METHOD Reset_Done : BOOL
VAR
	sTemp1 : T_MaxString;
END_VAR
IF sData = '' THEN
	Reset_Done := FALSE;
ELSE
	sTemp1 := sData;
	IF FC_Check_SOH(sTemp1) AND FC_Check_ACK(sTemp1) AND FC_Check_EOT(sTemp1) AND FC_Check_R(sTemp1) THEN
		Reset_Done := TRUE;
	ELSE
		Reset_Done := FALSE;
	END_IF
END_IF
END_METHOD

METHOD Start : BOOL
// Description : Ask for the status of the machine
VAR_INPUT
END_VAR
VAR
	sTemp1 : STRING;
	sTemp2 : STRING;
END_VAR
sData := '';
sTemp1 := 'S';
sTemp2 := CONCAT(SOH, sTemp1);
sCmd := CONCAT(sTemp2, EOT);
THIS^.Send(sCmd);
END_METHOD

METHOD Start_Done : BOOL
VAR
	sTemp1 : T_MaxString;
END_VAR
IF sData = '' THEN
	Start_Done := FALSE;
ELSE
	sTemp1 := sData;
	IF FC_Check_SOH(sTemp1) AND FC_Check_ACK(sTemp1) AND FC_Check_EOT(sTemp1) AND FC_Check_S(sTemp1) THEN
		Start_Done := TRUE;
	ELSE
		Start_Done := FALSE;
	END_IF
END_IF
END_METHOD

END_FUNCTION_BLOCK

// ---- FBs/Ethernet/FB_EthDevice.TcPOU
FUNCTION_BLOCK FB_EthDevice
VAR_INPUT
	bEnable		: BOOL 			:= FALSE;				(* TRUE => enable client data exchange, FALSE => disable *)
	sSrvNetID	: T_AmsNetID	:= '';					(* TwinCAT TCP/IP server network address *)
	sRemoteHost	: T_IPv4Addr 	:= '127.0.0.1';			(* Server network address *)
	nRemotePort	: UDINT 		:= 200;					(* Server port number *)
	bLogEnable	: BOOL 			:= FALSE;				(* TRUE => Enable log message output, FALSE => Disable *)
	sLogPrefix	: STRING 		:= 'CLIENT::';			(* Log message description string (allows the identification of log message source) *)
END_VAR
VAR_OUTPUT
	sData						: T_MaxString;			(* Output received Data *)
	bConnected					: BOOL := FALSE;		(* TCP/IP connection state *)	
END_VAR
VAR
	fbConnection				: FB_ClientConnection;	(* Client connection/data exchange control function block *)
	fbTx 						: FB_FrameFifo;			(* Tx fifo *)
	fbRx 						: FB_FrameFifo;			(* Rx fifo *)
	
	sLogMessage					: T_MaxString;
	sTemData					: T_MaxString;			(* Output received Data *)
END_VAR

IF bConnected := fbConnection.bConnected THEN
	A_Receive();
END_IF

A_Call();

IF NOT fbConnection.RxBusy THEN
	sData := sTemData;
END_IF

ACTION A_Call:
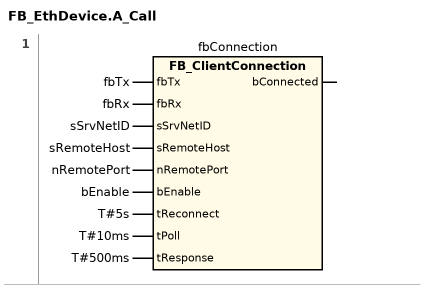
// NETWORK 1
fbConnection(
    fbTx := fbTx,
    fbRx := fbRx,
    sSrvNetID := sSrvNetID,
    sRemoteHost := sRemoteHost,
    nRemotePort := nRemotePort,
    bEnable := bEnable,
    tReconnect := T#5s,
    tPoll := T#10ms,
    tResponse := T#500ms); // FB_ClientConnection
END_ACTION

ACTION A_Receive:
	(*--------------------- Get received message strings --------------------------------*)
	REPEAT
		fbRx.RemoveHead( );(* Fetch string from rx fifo *)
		IF fbRx.bOk THEN(* Success *)
	
		(* TODO: Implement receive data handler *)
			sTemData := fbRx.sGet; 		
			
		END_IF
	UNTIL NOT fbRx.bOk
	END_REPEAT
END_ACTION

METHOD Send : BOOL
VAR_INPUT
	sTxData		: T_MaxString;	(* Data to send *)
END_VAR
VAR
	RTRIG_SendCommand			: R_TRIG;
END_VAR
		fbTx.AddTail( sPut := sTxData );(* Put string to the tx fifo *)
END_METHOD

END_FUNCTION_BLOCK

// ---- FBs/Ethernet/FB_ClientConnection.TcPOU
FUNCTION_BLOCK FB_ClientConnection
VAR_IN_OUT
	fbTx 			: FB_FrameFifo;(* TX fifo *)
	fbRx 			: FB_FrameFifo;(* RX fifo *)
END_VAR
VAR_INPUT
	sSrvNetID		: T_AmsNetID 	:= '';(* TwinCAT TCP/IP server network address *)
	sRemoteHost		: T_IPv4Addr 	:= '127.0.0.1';(* IP adress of remote server *)
	nRemotePort		: UDINT 		:= 0;(* Server port number *)
	bEnable			: BOOL 			:= FALSE;(* TRUE => connect and exchange data, FALSE => disconnect *)
	tReconnect 		: TIME 			:= T#5S;(* Try to reconnect after this time *)
	tPoll			: TIME 			:= T#50MS;(* Polling time *)
	tResponse		: TIME 			:= T#1S;(* Timeout waiting for response *)
END_VAR
VAR_OUTPUT
	bConnected		: BOOL 			:= FALSE;(* Established connection status *)
END_VAR
VAR
	fbConnect 		: FB_SocketConnect;
	fbClose			: FB_SocketClose;
	fbSend			: FB_SocketSend;
	fbReceive		: FB_SocketReceive;
	eStep			: eConnectionSteps;
	bSndBusy 		: BOOL;(* Tx state *)
	bRcvBusy 		: BOOL;(* Rx state *)
	bDisconnect		: BOOL;(* Disconnect flag, if set the socket will be closed *)
	
	TON_PollTimer		: TON;(* Receive poll timer *)
	TON_ResponseTimer 	: TON;(* Waiting response timeout timer *)
	TON_ReconnectTimer	: TON := (PT := T#5S);(* Reconnect timer *)
	
	rxBuffer			: ARRAY[0..PLCPRJ_BUFFER_SIZE] OF BYTE;
	sTxFrame			: T_MaxString;
	sRxFrame			: T_MaxString;
	cbReceived			: UDINT;
	nLenOfString		: UDINT;(* String length inclusive the null delimiter *)
	bEndOfString		: BOOL := FALSE;
	StartPolling		: BOOL; // 1 = reciving mode, polling reciving command until there is no new data in the socket (nRecBytes = 0) / 0 = reciving finished, send command again possible
	MemFirstFrame		: BOOL; // received at least one frame
	RxBusy				: BOOL; // received at least one frame
	RTRIG_FirstFrame	: R_TRIG; // trigger first frame
END_VAR

IF eStep <> eCONNECTION_STATE_DATAEXCHANGE THEN
	StartPolling 	:= FALSE;
	MemFirstFrame	:= FALSE;
	bRcvBusy 		:= FALSE;	
END_IF

CASE eStep OF
	eCONNECTION_STATE_IDLE:
		IF bEnable XOR bConnected THEN
			IF bEnable THEN
				TON_ReconnectTimer( IN := TRUE);
				IF TON_ReconnectTimer.Q THEN

					fbTx.Clear();(* Clear send fifo *)
					fbRx.Clear();(* Clear receiver fifo *)
					
					bSndBusy := FALSE;
					bRcvBusy := FALSE;
					bDisconnect := FALSE;
					cbReceived := 0;

					
					TON_ReconnectTimer( IN := FALSE, PT := tReconnect );

					eStep := eCONNECTION_STATE_CONNECT_START;
				END_IF
			ELSE
				eStep := eCONNECTION_STATE_CLOSE_START;
			END_IF
		ELSIF bConnected THEN
			eStep := eCONNECTION_STATE_DATAEXCHANGE;
		ELSE
			TON_ReconnectTimer( IN := FALSE, PT := T#0S );
		END_IF

	eCONNECTION_STATE_CONNECT_START:
		fbConnect( bExecute := FALSE );
		fbConnect( sSrvNetID := sSrvNetID, 
					sRemoteHost := sRemoteHost, 
					nRemotePort := nRemotePort, 
					bExecute := TRUE );
		eStep := eCONNECTION_STATE_CONNECT_WAIT;

	eCONNECTION_STATE_CONNECT_WAIT:
		fbConnect( bExecute := FALSE );
		IF NOT fbConnect.bBusy THEN
			IF NOT fbConnect.bError THEN
				bConnected 	:= TRUE;
				eStep := eCONNECTION_STATE_IDLE;
			ELSE
				
				eStep := eCONNECTION_STATE_ERROR;
			END_IF
		END_IF

	eCONNECTION_STATE_DATAEXCHANGE:
		TON_ResponseTimer(PT := PLCPRJ_RECEIVE_TIMEOUT);(* Bytes received => disable timeout check *)
		TON_PollTimer( IN := NOT TON_PollTimer.Q, PT := PLCPRJ_RECEIVE_POLLING_TIME );
		
		bDisconnect := NOT bEnable OR bDisconnect;(* User/internal disconnect requested? *)
		IF bDisconnect AND NOT bSndBusy AND NOT bRcvBusy THEN
			bDisconnect := FALSE;
			eStep := eCONNECTION_STATE_CLOSE_START;(* Disconnect *)
		ELSE
	
(* SEND *)
			IF NOT bDisconnect AND NOT bSndBusy AND NOT StartPolling THEN
				fbTx.RemoveHead( sGet => sTxFrame );(* Remove oldest string entry s*)
				IF fbTx.bOk THEN(* Success *)
					fbSend( bExecute := FALSE );
					fbSend(	sSrvNetID := sSrvNetID,
							hSocket	:= fbConnect.hSocket,
							pSrc	:= ADR( sTxFrame ),
							cbLen	:= INT_TO_UDINT(LEN( sTxFrame )) + 1,(* String length inclusive the zero delimiter *)
							bExecute:= TRUE ); // Send command
					bSndBusy := TRUE;
					StartPolling	:= FALSE;
				END_IF
			ELSE 
				fbSend( bExecute := FALSE );
				IF NOT fbSend.bBusy THEN
					// after send command
					bSndBusy := FALSE;
					IF fbSend.bError THEN
						
						bDisconnect := TRUE;(* Set flag *)
					END_IF
					
					IF NOT StartPolling THEN
						// start reciving until there is no new data in the socket or timeout
						TON_ResponseTimer.IN := TRUE;
						StartPolling	:= TRUE;
					END_IF;
				END_IF
			END_IF

(* RECEIVE *)
			RTRIG_FirstFrame( CLK := fbReceive.nRecBytes <> 0);
			IF RTRIG_FirstFrame.Q THEN
				// received at least one frame
				MemFirstFrame := TRUE;
			END_IF
			IF MemFirstFrame AND fbReceive.nRecBytes = 0 THEN
				// reciving finished
				StartPolling 	:= FALSE;
				MemFirstFrame	:= FALSE;
				bRcvBusy 		:= FALSE;
			END_IF
			IF NOT bDisconnect AND NOT bRcvBusy AND StartPolling THEN
				IF TON_PollTimer.Q THEN
					// polling
					fbReceive( bExecute := FALSE );
					fbReceive( 	sSrvNetID := sSrvNetID, 
								hSocket	:= fbConnect.hSocket,
								pDest	:= ADR( rxBuffer ) + cbReceived,
								cbLen	:= SIZEOF( rxBuffer ) - cbReceived,
								bExecute:= TRUE ); // Reciving command
					bRcvBusy := TRUE;
				END_IF
			ELSE
				fbReceive( bExecute := FALSE );
				IF NOT fbReceive.bBusy THEN
					// after reciving command
					bRcvBusy := FALSE;
					IF NOT fbReceive.bError THEN
						IF (fbReceive.nRecBytes > 0) THEN(* Bytes received *)
							TON_PollTimer( IN := FALSE, PT := T#0S ); (* Bytes received => increase the read (polling) speed *)
							TON_ResponseTimer.IN := FALSE;(* Bytes received => disable timeout check *)
							cbReceived 	:= cbReceived + fbReceive.nRecBytes;(* Calculate the number of received data bytes *)

							REPEAT
								
								(* Search for string end delimiter *)
								nLenOfString := 0;(* Reset string length *)
								bEndOfString := FALSE;
								REPEAT 
									IF rxBuffer[nLenOfString] = 0 THEN(* String end delimiter found *)
										bEndOfString := TRUE;
									END_IF
									nLenOfString := nLenOfString + 1;
								UNTIL bEndOfString OR (nLenOfString >= cbReceived)
								END_REPEAT
								
								IF bEndOfString OR (nLenOfString >= cbReceived) THEN
									MEMSET( ADR( sRxFrame ), 16#0, SIZEOF( sRxFrame ) );
									MEMCPY(  ADR( sRxFrame ), ADR( rxBuffer ), MIN( SIZEOF(sRxFrame), nLenOfString ) );(* Copy the received string to the output variable (inclusive the end delimiter) *)
									MEMMOVE( ADR( rxBuffer ), ADR( rxBuffer[nLenOfString] ), cbReceived - nLenOfString  );(* Move the reamaining data bytes *)
									cbReceived := cbReceived - nLenOfString;(* Recalculate the reamaining data byte length *)
			
									fbRx.AddTail( sPut := sRxFrame );(* Put received message to the rx fifo *)
									IF NOT fbRx.bOk THEN

										bDisconnect := TRUE;(* Set flag *)
										RETURN;
									END_IF
								END_IF
								
							UNTIL NOT bEndOfString OR (cbReceived = 0)
							END_REPEAT
		
						ELSE(* No bytes received: reciving finished or timeout*)
							IF TON_ResponseTimer.Q THEN (* Timeout error*)
								StartPolling 	:= FALSE;
								MemFirstFrame	:= FALSE;	
								
								TON_ResponseTimer.IN := FALSE;
								
								bDisconnect := TRUE;(* Set flag *)
							END_IF
						END_IF
						
					ELSE(* Receive error *)
						StartPolling 	:= FALSE;
						MemFirstFrame	:= FALSE;
						bRcvBusy 		:= FALSE;
												
						bDisconnect := TRUE;(* Set flag *)
					END_IF
				END_IF(* IF NOT fbReceive.bBusy THEN *)
				
			END_IF(* IF NOT bDisconnect AND NOT bRcvBusy THEN *)
		
		END_IF(* IF bDisconnect AND NOT bSndBusy AND NOT bRcvBusy THEN *)

(* DISCONNECT *)		
	eCONNECTION_STATE_CLOSE_START:
		
		TON_PollTimer.IN := FALSE;
		TON_ResponseTimer.IN := FALSE;
		//bForceRecive	:= FALSE;
		
		fbClose( bExecute := FALSE );
		fbClose( sSrvNetID := sSrvNetID, 
					hSocket:= fbConnect.hSocket, 
					bExecute:= TRUE );
		eStep := eCONNECTION_STATE_CLOSE_WAIT;

	eCONNECTION_STATE_CLOSE_WAIT:
		fbClose( bExecute := FALSE );
		IF NOT fbClose.bBusy THEN
			bConnected := FALSE;
			IF NOT fbClose.bError THEN
				eStep := eCONNECTION_STATE_IDLE;
			ELSE
				
				eStep := eCONNECTION_STATE_ERROR;
			END_IF
		END_IF

	eCONNECTION_STATE_ERROR:(* Error step *)
		IF bConnected THEN
			eStep := eCONNECTION_STATE_CLOSE_START;
		ELSE
			eStep := eCONNECTION_STATE_IDLE;
		END_IF
END_CASE
RxBusy := MemFirstFrame;

METHOD ForceRecive : BOOL
VAR_INPUT
END_VAR
TON_ResponseTimer.IN := TRUE;
StartPolling	:= TRUE;
END_METHOD

END_FUNCTION_BLOCK

// ---- FBs/Ethernet/FB_FrameFifo.TcPOU
(* Tx/Rx (string data) fifo control function block *)
FUNCTION_BLOCK FB_FrameFifo
VAR_INPUT
	sPut		: T_MaxString 	:= ''; (* String message to add (write) to the fifo *)
END_VAR
VAR_OUTPUT
	bOk			: BOOL; 	 	(* TRUE = New entry added or removed succesfully, FALSE = Fifo overflow or fifo empty *)
	sGet		: T_MaxString 	:= '';(* String message removed (read) from fifo *)
	nCount		: UDINT			:= 0;(* Number of fifo entries *)
	cbFree		: UDINT 		:= 0;(* Free buffer space *)
END_VAR
VAR
	fbBuffer 	: FB_StringRingBuffer := (bOverwrite := FALSE);(* Basic (lower level) string buffer control function block *)
	buffer		: ARRAY[-3..PLCPRJ_BUFFER_SIZE] OF BYTE;(* Internal buffer memory *)
END_VAR

;

ACTION AddTail:
(* Adds new fifo entry *)
fbBuffer.A_AddTail( pBuffer:= ADR(buffer), cbBuffer:= SIZEOF(buffer),
					putValue:= sPut, bOk=>bOk, nCount=>nCount );
IF bOk THEN
	
	cbFree := PLCPRJ_BUFFER_SIZE - fbBuffer.cbSize;(* Calculate the free buffer space *)
END_IF
END_ACTION

ACTION Clear:
(* Resets fifo = clears all data *)
fbBuffer.A_Reset( pBuffer:= ADR(buffer), cbBuffer:= SIZEOF(buffer),
				bOk=>bOk, getValue=>sGet, nCount=>nCount );
cbFree := PLCPRJ_BUFFER_SIZE;(* Free buffer size *)
END_ACTION

ACTION RemoveHead:
(* Removes oldest fifo entry *)
fbBuffer.A_RemoveHead( pBuffer:= ADR(buffer), cbBuffer:= SIZEOF(buffer),
						bOk=>bOk, getValue=>sGet, nCount=>nCount );
IF bOk THEN
	cbFree := PLCPRJ_BUFFER_SIZE - fbBuffer.cbSize;(* Calculate the free buffer space *)
END_IF
END_ACTION

END_FUNCTION_BLOCK

// ---- FBs/LaserMarker - LASIT/FC_Check_SOH.TcPOU
FUNCTION FC_Check_SOH : BOOL
VAR_INPUT
	I_sString : REFERENCE TO T_MaxString;
END_VAR
VAR
	stringPos	: INT;
END_VAR

stringPos := FIND(I_sString, SOH);
IF stringPos <> 0 THEN
	I_sString := MID(I_sString, LEN(I_sString), stringPos+1);
	FC_Check_SOH := TRUE;
ELSE
	FC_Check_SOH := FALSE;
END_IF

END_FUNCTION

// ---- FBs/LaserMarker - LASIT/FC_Check_ACK.TcPOU
FUNCTION FC_Check_ACK : BOOL
VAR_INPUT
	I_sString : REFERENCE TO T_MaxString;
END_VAR
VAR
	stringPos	: INT;
END_VAR

stringPos := FIND(I_sString, ACK);
IF stringPos <> 0 THEN
	I_sString := MID(I_sString, LEN(I_sString), stringPos+1);
	FC_Check_ACK := TRUE;
ELSE
	FC_Check_ACK := FALSE;
END_IF

END_FUNCTION

// ---- FBs/LaserMarker - LASIT/FC_Check_EOT.TcPOU
FUNCTION FC_Check_EOT : BOOL
VAR_INPUT
	I_sString : REFERENCE TO T_MaxString;
END_VAR
VAR
	stringPos	: INT;
END_VAR

stringPos := FIND(I_sString, EOT);
IF stringPos <> 0 THEN
	I_sString := MID(I_sString, stringPos-1, 1);
	FC_Check_EOT := TRUE;
ELSE
	FC_Check_EOT := FALSE;
END_IF

END_FUNCTION

// ---- FBs/LaserMarker - LASIT/FC_Check_T.TcPOU
FUNCTION FC_Check_T : BOOL
VAR_INPUT
	I_sString : REFERENCE TO T_MaxString;
END_VAR
VAR
	stringPos	: INT;
END_VAR

stringPos := FIND(I_sString, 'T');
IF stringPos <> 0 THEN
	I_sString := MID(I_sString, LEN(I_sString), stringPos+1);
	FC_Check_T := TRUE;
ELSE
	FC_Check_T := FALSE;
END_IF

END_FUNCTION

// ---- FBs/LaserMarker - LASIT/FC_Check_IN.TcPOU
FUNCTION FC_Check_IN : BOOL
VAR_INPUT
	I_sString : REFERENCE TO T_MaxString;
END_VAR
VAR
	stringPos	: INT;
END_VAR

stringPos := FIND(I_sString, 'IN');
IF stringPos <> 0 THEN
	I_sString := MID(I_sString, LEN(I_sString), stringPos+1);
	FC_Check_IN := TRUE;
ELSE
	FC_Check_IN := FALSE;
END_IF

END_FUNCTION

// ---- FBs/LaserMarker - LASIT/FC_Check_J.TcPOU
FUNCTION FC_Check_J : BOOL
VAR_INPUT
	I_sString : REFERENCE TO T_MaxString;
END_VAR
VAR
	stringPos	: INT;
END_VAR

stringPos := FIND(I_sString, 'J');
IF stringPos <> 0 THEN
	I_sString := MID(I_sString, LEN(I_sString), stringPos+1);
	FC_Check_J := TRUE;
ELSE
	FC_Check_J := FALSE;
END_IF

END_FUNCTION

// ---- FBs/LaserMarker - LASIT/FC_Check_K.TcPOU
FUNCTION FC_Check_K : BOOL
VAR_INPUT
	I_sString : REFERENCE TO T_MaxString;
END_VAR
VAR
	stringPos	: INT;
END_VAR

stringPos := FIND(I_sString, 'K');
IF stringPos <> 0 THEN
	I_sString := MID(I_sString, LEN(I_sString), stringPos+1);
	FC_Check_K := TRUE;
ELSE
	FC_Check_K := FALSE;
END_IF

END_FUNCTION

// ---- FBs/LaserMarker - LASIT/FC_Check_R.TcPOU
FUNCTION FC_Check_R : BOOL
VAR_INPUT
	I_sString : REFERENCE TO T_MaxString;
END_VAR
VAR
	stringPos	: INT;
END_VAR

stringPos := FIND(I_sString, 'R');
IF stringPos <> 0 THEN
	I_sString := MID(I_sString, LEN(I_sString), stringPos+1);
	FC_Check_R := TRUE;
ELSE
	FC_Check_R := FALSE;
END_IF

END_FUNCTION

// ---- FBs/LaserMarker - LASIT/FC_Check_S.TcPOU
FUNCTION FC_Check_S : BOOL
VAR_INPUT
	I_sString : REFERENCE TO T_MaxString;
END_VAR
VAR
	stringPos	: INT;
END_VAR

stringPos := FIND(I_sString, 'S');
IF stringPos <> 0 THEN
	I_sString := MID(I_sString, LEN(I_sString), stringPos+1);
	FC_Check_S := TRUE;
ELSE
	FC_Check_S := FALSE;
END_IF

END_FUNCTION

// ---- FBs/LaserMarker - LASIT/FB_FlyPowerMarkManager.TcPOU
FUNCTION_BLOCK FB_FlyPowerMarkManager
VAR_INPUT
	In : BOOL;
END_VAR
VAR_OUTPUT
	Out : BOOL;
END_VAR
VAR
	RTRIG_Enable	: R_TRIG;
	TON_DelayEnable	: TON;
END_VAR

TON_DelayEnable(IN := In, PT := T#1S);	
RTRIG_Enable(CLK := TON_DelayEnable.Q);

IF RTRIG_Enable.Q THEN
	Out := TRUE;
ELSIF NOT TON_DelayEnable.Q THEN
	Out := FALSE;
END_IF

END_FUNCTION_BLOCK

// ---- FBs/LaserMarker - LASIT/FB_FlyPowerMarkExeManager.TcPOU
FUNCTION_BLOCK FB_FlyPowerMarkExeManager
VAR_INPUT
	UpsPowerStatus : E_UpsPowerStatus;
	LasitControllerOn : BOOL;
	Reset : BOOL;
END_VAR
VAR_OUTPUT
	Error	: BOOL  := FALSE;
	ErrorID	: INT 	:= 0;
	ErrorSubID	: INT 	:= 0;
END_VAR
VAR_IN_OUT
	Init	: BOOL;
	NT_OpenExe : NT_StartProcess;
	NT_CloseExe : NT_StartProcess;
END_VAR
VAR
	iState				: INT 	:= 0;
	RTRIG_PowerOnLine	: R_TRIG;
	RTRIG_PowerOnBattery	: R_TRIG;
	RTRIG_Reset			: R_TRIG;
	DelayOpenExe		: TON;
	TON_Timeout			: TON;
	tTimeout			: TIME := T#10S;
END_VAR

RTRIG_PowerOnLine(CLK := UpsPowerStatus = E_UpsPowerStatus.PowerOnLine);
RTRIG_PowerOnBattery(CLK := UpsPowerStatus = E_UpsPowerStatus.PowerOnBattery);

RTRIG_Reset(CLK := Reset);
IF RTRIG_Reset.Q THEN
	iState := 0;
	ErrorID 	:= 0;
	ErrorSubID := 0;
	Error		:= FALSE;
END_IF

IF RTRIG_PowerOnLine.Q THEN
	NT_OpenExe.START := FALSE;
	NT_CloseExe.START := FALSE;
	iState := 10;
END_IF

IF RTRIG_PowerOnBattery.Q THEN
	NT_OpenExe.START := FALSE;
	NT_CloseExe.START := FALSE;
	iState := 100;
END_IF

DelayOpenExe(IN := iState = 10 AND LasitControllerOn, PT := T#30S);

CASE iState OF
	0:
		;
		
	10:
		IF Init THEN
			Init := FALSE;
			iState := 0;
		ELSIF DelayOpenExe.Q THEN
			//NT_OpenExe.COMNDLINE := 'FLY_POWERMARK.exe "C:\Program Files (x86)\Lasit spa\Laser_FLY_POWERMARK\FLY_POWERMARK.exe"'; 
			//togliere commento se si vuole attivare debug dell'esecuzione del .bat
			NT_OpenExe.COMNDLINE := 'FLY_POWERMARK.exe "C:\Program Files (x86)\Lasit spa\Laser_FLY_POWERMARK\FLY_POWERMARK.exe" debug'; 
		
			iState := 20;
		END_IF
		
	20:
		NT_OpenExe.START := TRUE;
		IF NT_OpenExe.BUSY THEN
			iState := 30;
		END_IF
		
	30:
		IF NOT NT_OpenExe.BUSY THEN
			NT_OpenExe.START := FALSE;
			iState := 0;
		ELSIF NT_OpenExe.ERR THEN
			NT_OpenExe.START := FALSE;
			iStateError();
		END_IF		

	100:
		//NT_CloseExe.COMNDLINE := 'FLY_POWERMARK.exe';
		//togliere commento se si vuole attivare debug dell'esecuzione del .bat
		NT_CloseExe.COMNDLINE := 'FLY_POWERMARK.exe debug';
		iState := 110;
		
	110:
		NT_CloseExe.START := TRUE;
		IF NT_CloseExe.BUSY THEN
			iState := 120;
		END_IF
		
	120:
		IF NOT NT_CloseExe.BUSY THEN
			NT_CloseExe.START := FALSE;
			iState := 0;
		ELSIF NT_CloseExe.ERR THEN
			NT_CloseExe.START := FALSE;
			iStateError();
		END_IF		
	
END_CASE

//Timeout
Timeout();

// ERROR
ErrorSet();

METHOD PRIVATE ErrorSet : BOOL
IF (iState >= 1000) THEN
	ErrorID 	:= iState;
	Error		:= TRUE;
	ErrorSet	:= TRUE;
	
	iState		:= -1;
ELSE
	ErrorSet := FALSE;
END_IF
END_METHOD

METHOD PRIVATE iStateError
iState := iState + 1000;
END_METHOD

METHOD PRIVATE Timeout : BOOL
TON_Timeout(IN:= iState > 0 AND iState < 1000 AND iState <> 10 AND tTimeout <> T#0MS, PT := tTimeout);
IF TON_Timeout.Q THEN
    ErrorSubID := iState;
	Timeout := TRUE;
	
    iState := 1999;
ELSE
	Timeout := FALSE;
END_IF
END_METHOD

END_FUNCTION_BLOCK

// ---- FBs/FB_DataBufferManager.TcPOU
FUNCTION_BLOCK PUBLIC FB_DataBufferManager
VAR_INPUT
	ArraySize : INT;
	DataRepository : POINTER TO DataBuffer;	 // Element 0 for data preparation
END_VAR

METHOD Clear : BOOL
VAR_INPUT
	Position : INT := -1;
END_VAR
	IF (Position>0 AND Position<ArraySize) THEN
// Clear single position array repository  
		MEMSET(ADR(DataRepository[Position]), 16#00, SIZEOF(DataBuffer));
	ELSIF Position =-1 THEN
// Clear all position array	repository	
		MEMSET(ADR(DataRepository), 16#00, SIZEOF(DataRepository));
	ELSE
// Error
		;
	END_IF
END_METHOD

METHOD Ins : BOOL
VAR_INPUT
	DataIn: DataBuffer;
END_VAR
VAR
	i: UINT;
END_VAR
;
(*IF NOT DataRepository[0].PartState.Valid THEN
	MEMCPY(ADR(DataRepository[0]), ADR(DataIn), SIZEOF(DUT_PartData));	
ELSE
	// Error: GetNewPartData called with slot 0 non empty
END_IF*)

MEMCPY(ADR(DataRepository[0]), ADR(DataIn), SIZEOF(DataBuffer));
END_METHOD

METHOD M_Move : BOOL
VAR_INPUT
	DestPos		: UINT;
	SourcePos	: UINT;
END_VAR
IF DestPos >= 0 AND DestPos <= ArraySize AND SourcePos >=0 AND SourcePos <= ArraySize THEN
	MEMCPY(ADR(DataRepository[DestPos]), ADR(DataRepository[SourcePos]), SIZEOF(DataBuffer));
	
	MEMSET(ADR(DataRepository[SourcePos]), 16#00, SIZEOF(DataBuffer));
ELSE
	;//error
END_IF
END_METHOD

METHOD PUBLIC Read : BOOL
VAR_INPUT
	Position 	: UINT;
END_VAR

VAR_OUTPUT
	Dest		: DataBuffer;
END_VAR

//CASE Position OF
//	0..NUM_STAIONS:
//		MEMCPY(ADR(Dest), ADR(DataRepository[Position]), SIZEOF(DUT_PartData));
//ELSE	
//	;	// Error
//END_CASE

IF (Position>0 AND Position<20) THEN
		MEMCPY(ADR(Dest), ADR(DataRepository[Position]), SIZEOF(DataBuffer));
ELSE	
	;	// Error
END_IF
END_METHOD

METHOD PUBLIC Shift : BOOL
VAR
	i : UINT;
END_VAR
// Shift data array from StartPos(first data array moved) to EndPos (Last data array destination)
FOR i:= ArraySize TO 1 BY -1 DO
	MEMCPY(ADR(DataRepository[i]), ADR(DataRepository[i-1]), SIZEOF(DataBuffer));
END_FOR;

// Clear start position data array
MEMSET(ADR(DataRepository[0]), 16#00, SIZEOF(DataBuffer));
END_METHOD

METHOD PUBLIC ShiftRange : BOOL
VAR_INPUT
	StartPos	: INT;
	EndPos 		: INT;
END_VAR
VAR
	i : INT;
	N : INT := 0;
END_VAR
IF(StartPos < EndPos AND EndPos <= ArraySize) THEN
	N := EndPos - StartPos - 1;
	FOR i:= 0 TO N DO
		MEMCPY(ADR(DataRepository[EndPos-i]), ADR(DataRepository[EndPos-i-1]), SIZEOF(DataBuffer));
	END_FOR;
ELSE
	; //Error;
END_IF;

// Clear start position data array
MEMSET(ADR(DataRepository[StartPos]), 16#00, SIZEOF(DataBuffer));
END_METHOD

METHOD Update : BOOL
VAR_INPUT
END_VAR
// TODO: GraphQL mutation with FIFO
END_METHOD

END_FUNCTION_BLOCK

// ---- FBs/DataRequest/FB_DataRequest.TcPOU
FUNCTION_BLOCK FB_DataRequest
VAR_INPUT
	Reset			: BOOL;
	ExecuteCurrent  : BOOL;
	ExecuteNext		: BOOL; 
	WID				: DWORD;
	MachineEmpty	: BOOL;
END_VAR
VAR_OUTPUT
	Done			: BOOL;
	Busy			: BOOL;
	Error			: BOOL;
	ErrorID			: DINT;
	ErrorSubID		: DINT;
	Elapsed			: TIME;
	ErrorCodePMC	: BYTE;
END_VAR
VAR_IN_OUT
	St0Data : DUT_St0Data;
	fbShiftDataBuffer		: FB_DataBufferManager;
	WID_Old			: DINT;
	PMC_ShiftManData0 		: stShiftData;
END_VAR
VAR
	i				: UDINT;
	iState			: INT := -1;
	RTRIG_ReqNext	: R_TRIG;
	RTRIG_Reset	: R_TRIG;
	RTRIG_Empty		: R_TRIG;
	FTRIG_Empty		: F_TRIG;
	TON_Elaspse		: TON;
	Next			: BOOL;
	TempDataBuffer 		: DataBuffer;
	memEmpty		: BOOL;
	tempstByteAsBit	: stByteAsBit;
END_VAR

IF NOT ExecuteCurrent AND NOT ExecuteNext AND iState = 1030 THEN
	iState := -1;
END_IF

RTRIG_Reset(CLK:=Reset);
IF RTRIG_Reset.Q AND Error THEN
	Error := FALSE; // Error
	ErrorID := 0;
	ErrorSubID := 0;
	iState := -1;
END_IF

RTRIG_ReqNext(CLK := ExecuteCurrent OR ExecuteNext); // Request
TON_Elaspse(IN:= Busy, PT:=T#10S);
IF TON_Elaspse.Q THEN
	ErrorSubID := iState;
	iState := 1999;
END_IF
IF RTRIG_ReqNext.Q AND NOT Busy THEN
	Next := ExecuteNext;
	Error := FALSE; // Error
	ErrorID := 0;
	ErrorSubID := 0;
	iState := 0;
END_IF

RTRIG_Empty(CLK := MachineEmpty AND NOT Busy);
IF RTRIG_Empty.Q THEN
	memEmpty := TRUE;
	IF Error THEN
		Error := FALSE;
		ErrorID := 0;
		ErrorSubID := 0;
	END_IF
END_IF
FTRIG_Empty(CLK := MachineEmpty);
IF FTRIG_Empty.Q THEN
	memEmpty := FALSE;
END_IF
IF memEmpty AND ErrorID = 1030 THEN
	Error := FALSE; // Error
	ErrorCodePMC := 0;
END_IF

CASE iState OF
	-1:
		Done := FALSE; // Done
		Busy := FALSE; // Busy
	
	0:
		Error := FALSE; // Error
		MEMSET(ADR(St0Data), 0, SIZEOF(St0Data));
		PMC_ShiftManData0.FLAGP.aBit.b0 := FALSE;
		ErrorCodePMC := 0;
		Busy := TRUE;
		
		IF WID<>0 THEN
			IF WID_Old <> DWORD_TO_DINT(St0Data.WindP) OR WID_Old <> DWORD_TO_DINT(WID) THEN
				iState := 10;
			ELSE		
				iState := 997;
			END_IF	
		ELSE		
			iState := 10;
		END_IF		
		
	10:
		PRG_MSSQL_spGetNextPartPLCData.Execute := TRUE;
		IF PRG_MSSQL_spGetNextPartPLCData.Busy THEN
			
			iState := 20;
		END_IF
		
	20:
		IF PRG_MSSQL_spGetNextPartPLCData.Done THEN
			
			iState := 30;
		ELSIF PRG_MSSQL_spGetNextPartPLCData.Error THEN
			PRG_MSSQL_spGetNextPartPLCData.Execute := FALSE;
			
			iState := 1020;
		END_IF
		
	30:
		IF PRG_MSSQL_spGetNextPartPLCData.DataGood THEN 
			PRG_MSSQL_spGetNextPartPLCData.Execute := FALSE;
	
			tempstByteAsBit.aByte := 0;
			tempstByteAsBit.aBit.b0 := SEL(STRING_TO_INT(DB.stPLCData.IsFirstPartInBatch) = 1, FALSE, TRUE);
			tempstByteAsBit.aBit.b1 := SEL(STRING_TO_INT(DB.stPLCData.IsLastPartInBatch) = 1, FALSE, TRUE);
			tempstByteAsBit.aBit.b2 := SEL(STRING_TO_INT(DB.stPLCData.IsFirstPartInRow) = 1, FALSE, TRUE);
			tempstByteAsBit.aBit.b3 := SEL(STRING_TO_INT(DB.stPLCData.IsLastPartInRow) = 1, FALSE, TRUE);			
			St0Data.FlagP[2] := tempstByteAsBit.aByte;
			
			St0Data.WindP := SEL(Next, WID, DINT_TO_DWORD(DB.stPLCData.PartId));
			St0Data.TpcyS[3]  := DINT_TO_BYTE(DB.stPLCData.BroachingPlan.PassCount);		

			// Giro 1
			FC_BroachingPlanCopyPass(ADR(St0Data.TpcyS[5]), DB.stPLCData.BroachingPlan.Pass1BaseBroachingPlan, DB.stPLCData.BroachingPlan.Pass1VariantsBroachingPlan);		
			// Giro 2
			FC_BroachingPlanCopyPass(ADR(St0Data.TpcyS[12]), DB.stPLCData.BroachingPlan.Pass2BaseBroachingPlan, DB.stPLCData.BroachingPlan.Pass2VariantsBroachingPlan);			
			// Giro 3
			FC_BroachingPlanCopyPass(ADR(St0Data.TpcyS[19]), DB.stPLCData.BroachingPlan.Pass3BaseBroachingPlan, DB.stPLCData.BroachingPlan.Pass3VariantsBroachingPlan);		
			// Giro 4  
			FC_BroachingPlanCopyPass(ADR(St0Data.TpcyS[26]), DB.stPLCData.BroachingPlan.Pass4BaseBroachingPlan, DB.stPLCData.BroachingPlan.Pass4VariantsBroachingPlan);       	

			// Tipo di sbavatura
			tempstByteAsBit.aByte := 0;
			tempstByteAsBit.aBit.b0 := SEL(DB.stPLCData.Brushing = '5Pins', FALSE, TRUE);
			tempstByteAsBit.aBit.b1 := SEL(DB.stPLCData.Brushing = '6Pins', FALSE, TRUE);
			St0Data.TpcyS[33] := tempstByteAsBit.aByte;
			
			// sbavatura foro coda si, no
			IF DB.stPLCData.BackHole = '' THEN
				// errore stringa abilitazione foro coda
				St0Data.TpcyS[34] := 0;
				iState := 1031;
				RETURN;
			ELSIF DB.stPLCData.BackHole = 'No' THEN
				St0Data.TpcyS[34] := 0;
			ELSIF DB.stPLCData.BackHole = 'Si' THEN
				St0Data.TpcyS[34] := 1; 
			ELSE
				// errore stringa abilitazione foro coda
				St0Data.TpcyS[34] := 0;
				iState := 1032;
				RETURN;
			END_IF
			
			// tipo di scarico
			St0Data.TpcyS[35] :=DINT_TO_BYTE(DB.stPLCData.UnloadingModeId);
			
			FC_BroachingPlanCopyConpensation(ADR(St0Data.Data[1]), DB.stPLCData.BroachingPlan.Pass1BaseBroachingPlan, DB.stPLCData.BroachingPlan.Pass1VariantsBroachingPlan);	
			// Giro 1		
			FC_BroachingPlanCopyConpensation(ADR(St0Data.Data[1]), DB.stPLCData.BroachingPlan.Pass1BaseBroachingPlan, DB.stPLCData.BroachingPlan.Pass1VariantsBroachingPlan);
			// Giro 2
			FC_BroachingPlanCopyConpensation(ADR(St0Data.Data[22]), DB.stPLCData.BroachingPlan.Pass2BaseBroachingPlan, DB.stPLCData.BroachingPlan.Pass2VariantsBroachingPlan);		
			// Giro 3
			FC_BroachingPlanCopyConpensation(ADR(St0Data.Data[43]), DB.stPLCData.BroachingPlan.Pass3BaseBroachingPlan, DB.stPLCData.BroachingPlan.Pass3VariantsBroachingPlan);		
			// Giro 4
			FC_BroachingPlanCopyConpensation(ADR(St0Data.Data[64]), DB.stPLCData.BroachingPlan.Pass4BaseBroachingPlan, DB.stPLCData.BroachingPlan.Pass4VariantsBroachingPlan);			
			
			iState := 997;
		ELSIF PRG_MSSQL_spGetNextPartPLCData.Empty THEN
			PRG_MSSQL_spGetNextPartPLCData.Execute := FALSE;
			St0Data.WindP := 0;
			PMC_ShiftManData0.WIDP := DWORD_TO_DINT(St0Data.WindP);
			
			iState := 1030;
		END_IF
		
	997:
		PMC_ShiftManData0.WIDP := DWORD_TO_DINT(St0Data.WindP);
		TempDataBuffer.WIDP				:= DWORD_TO_DINT(St0Data.WindP);
		TempDataBuffer.PmcData				:= St0Data;
		TempDataBuffer.stPLCData			:= DB.stPLCData;
		PMC_ShiftManData0.FLAGP.aBit.b0 := TRUE;	
	
		fbShiftDataBuffer.Ins(TempDataBuffer);
		WID_Old := DWORD_TO_DINT(WID);
		
		Done := TRUE;
		Busy := FALSE;
		Elapsed := TON_Elaspse.ET;
		
		iState := 998;
		
	998:
		fbShiftDataBuffer.Shift();
		iState := 999;
		
	999:
		IF NOT ExecuteCurrent AND NOT ExecuteNext THEN
			iState := -1;
		END_IF
	
END_CASE

IF(iState > 999) THEN
	Done			:= FALSE;
	Busy			:= FALSE;
	Error			:= TRUE;
	ErrorID := iState;
	ErrorCodePMC := SEL(ErrorID = 1030, SINT_TO_BYTE(-1), SINT_TO_BYTE(1));
END_IF

END_FUNCTION_BLOCK

// ---- FBs/Database/PRG_MSSQL_spGetNextPartPLCData.TcPOU
PROGRAM PRG_MSSQL_spGetNextPartPLCData
VAR_INPUT
	Execute					: BOOL;
	Enable					: BOOL;
	OtherSPBusy				: BOOL;
END_VAR
VAR_OUTPUT
	Error					: BOOL;
	ErrorID					: DINT;
	Done					: BOOL;
	Busy					: BOOL;
	tcMessage 				: I_TcMessage;
	Q_tElapsedTime			: TIME;
	Buffer					: STRING(DB.MAX_STRING_SIZE);
	DataGood				: BOOL;
	Empty					: BOOL;
END_VAR
VAR
	RTRIG_Execute			: R_TRIG;
	iState					: INT := -1;
	fbJsonDataType 			: FB_JsonReadWriteDataType;
	Parameters				: DUT_NextPartPLCData;
	NumRetry				: USINT;
	TON_DelayRetry			: TON;
END_VAR
VAR_IN_OUT
	fbSQLResult				: FB_SQLResultEvt;
	fbSQLStoredProcedure	: FB_SQLStoredProcedureEvt;
	stPLCData				: DUT_stPLCData;
END_VAR

TON_DelayRetry(IN := iState = 15, PT := T#200MS);
RTRIG_Execute(CLK := Execute AND Enable);
IF(RTRIG_Execute.Q) THEN
	 Done							:= FALSE;
	 Error							:= FALSE;
	 ErrorID						:= 0; 
	 
	 iState							:= 0;
ELSIF NOT Execute AND NOT Busy THEN
	Busy			:= FALSE;
	Done			:= FALSE;
	Error			:= FALSE;
	Empty								:= FALSE;
	DataGood 							:= FALSE;
	
	iState := -1;
END_IF
 
 CASE iState OF
 
	 0:
		Busy								:= TRUE;
		NumRetry							:= 1;
		IF NOT OtherSPBusy THEN
			iState 								:= 10;
		END_IF
		
	10:
		//Buffer := '{"PartId":1,"RowIndex":"1","RunningNo":"1","ProfileName":"D0U12","FamilyName":"1200","PlugType":"3800.9","IsFirstPartInBatch":"1","IsLastPartInBatch":"0","IsFirstPartInRow":"1","IsLastPartInRow":"0","MarkingData":{"LayoutName":"Default","OrderReference":"PRD0000001","ProfileLaser":"D0U12"},"Brushing":"5Pins","BackHole":"No","UnloadingModeId":1,"BroachingPlan":{"PassCount":2,"Pass1BaseBroachingPlan":{"ToolHolderBase_Position":1,"ToolHolderBase_BroachName":"1200","ToolHolderBase_LateralCompensation":0.000,"ToolHolderBase_DepthCompensation":0.000,"ToolHolderBase_AngleCompensation":0.000},"Pass1VariantsBroachingPlan":{"ToolHolderA_Position":24,"ToolHolderA_BroachName":"___A","ToolHolderA_LateralCompensation":0.000,"ToolHolderA_DepthCompensation":0.000,"ToolHolderA_AngleCompensation":0.000,"ToolHolderB_Position":24,"ToolHolderB_BroachName":"___B","ToolHolderB_LateralCompensation":0.000,"ToolHolderB_DepthCompensation":0.000,"ToolHolderB_AngleCompensation":0.000,"ToolHolderC_Position":24,"ToolHolderC_BroachName":"___C","ToolHolderC_LateralCompensation":0.000,"ToolHolderC_DepthCompensation":0.000,"ToolHolderC_AngleCompensation":0.000,"ToolHolderD_Position":2,"ToolHolderD_BroachName":"U7","ToolHolderD_LateralCompensation":0.000,"ToolHolderD_DepthCompensation":0.000,"ToolHolderD_AngleCompensation":0.000,"ToolHolderE_Position":1,"ToolHolderE_BroachName":"U8","ToolHolderE_LateralCompensation":0.000,"ToolHolderE_DepthCompensation":0.000,"ToolHolderE_AngleCompensation":0.000,"ToolHolderF_Position":1,"ToolHolderF_BroachName":"D10","ToolHolderF_LateralCompensation":0.000,"ToolHolderF_DepthCompensation":0.000,"ToolHolderF_AngleCompensation":0.000},"Pass2BaseBroachingPlan":{"ToolHolderBase_Position":24,"ToolHolderBase_BroachName":"____","ToolHolderBase_LateralCompensation":0.000,"ToolHolderBase_DepthCompensation":0.000,"ToolHolderBase_AngleCompensation":0.000},"Pass2VariantsBroachingPlan":{"ToolHolderA_Position":2,"ToolHolderA_BroachName":"D20","ToolHolderA_LateralCompensation":0.000,"ToolHolderA_DepthCompensation":0.000,"ToolHolderA_AngleCompensation":0.000,"ToolHolderB_Position":24,"ToolHolderB_BroachName":"___B","ToolHolderB_LateralCompensation":0.000,"ToolHolderB_DepthCompensation":0.000,"ToolHolderB_AngleCompensation":0.000,"ToolHolderC_Position":24,"ToolHolderC_BroachName":"___C","ToolHolderC_LateralCompensation":0.000,"ToolHolderC_DepthCompensation":0.000,"ToolHolderC_AngleCompensation":0.000,"ToolHolderD_Position":4,"ToolHolderD_BroachName":"D50","ToolHolderD_LateralCompensation":0.000,"ToolHolderD_DepthCompensation":0.000,"ToolHolderD_AngleCompensation":0.000,"ToolHolderE_Position":2,"ToolHolderE_BroachName":"D60","ToolHolderE_LateralCompensation":0.000,"ToolHolderE_DepthCompensation":0.000,"ToolHolderE_AngleCompensation":0.000,"ToolHolderF_Position":24,"ToolHolderF_BroachName":"___F","ToolHolderF_LateralCompensation":0.000,"ToolHolderF_DepthCompensation":0.000,"ToolHolderF_AngleCompensation":0.000}}}';
		//iState := 40; 
		IF fbSQLStoredProcedure.ExecuteDataReturn(pParameterStrc := ADR(Parameters), cbParameterStrc := SIZEOF(Parameters), pSQLDBResult := ADR(fbSQLResult)) THEN
			IF fbSQLStoredProcedure.bError THEN
				tcMessage := fbSQLStoredProcedure.ipTcResult;
				NumRetry := NumRetry + 1;
				IF NumRetry > 3 THEN
					iState 							:= 1010; 
				ELSE
					iState 							:= 15; 
				END_IF
			ELSE
				IF Parameters.return_value = 0 THEN
					DataGood := TRUE;
					Empty := FALSE;
					
					iState 							:= 30; 
				ELSIF Parameters.return_value = 100 THEN
					Empty := TRUE;
					DataGood := FALSE;
					
					iState 							:= 999; 
				ELSE 				
					DataGood := FALSE;
					Empty := FALSE;
					IF Parameters.return_value < 0 THEN
						iState := -10000 + TO_INT(Parameters.return_value);
					ELSE
						iState := 10000 + TO_INT(Parameters.return_value);
					END_IF
				END_IF
			END_IF    
		END_IF
		
	15:
		IF TON_DelayRetry.Q THEN
			iState 							:= 10;
		END_IF
		
	20:
		IF fbSQLResult.Read(0, fbSQLResult.nDataCount, ADR(Buffer), SIZEOF(Buffer), FALSE, TRUE) THEN
			IF fbSQLResult.bError THEN
				iState 							:= 1020;
			ELSE
				
				iState 							:= 30;
			END_IF
		END_IF
		
	30:
		IF fbSQLResult.Release() THEN
			iState 								:= 40;		
		END_IF
		
	40:	
		IF(fbJsonDataType.SetSymbolFromJson(Parameters.PLCData,'DUT_stPLCData', SIZEOF(stPLCData), ADR(stPLCData))) THEN	
			
			iState 								:= 999;	
			
		ELSE
			iState 								:= 1040;
		END_IF			
	
	999:
		Done			:= TRUE;
		Busy			:= FALSE;
		
 END_CASE 
 
IF iState > 1000 OR iState <= -10000 THEN
	Error 		:= TRUE;
	ErrorID	 	:= iState; 
	Busy	 	:= FALSE;
	iState := -1;
END_IF

END_PROGRAM

// ---- FBs/DataRequest/FC_BroachingPlanCopyPass.TcPOU
FUNCTION FC_BroachingPlanCopyPass
VAR_INPUT
	pByte : POINTER TO BYTE;
	BaseBroachingPlan 		: DUT_stBroachingPlanBase;     
    VariantsBroachingPlan	: DUT_stBroachingPlanVariants;
END_VAR

pByte[0]	:= DINT_TO_BYTE(BaseBroachingPlan.ToolHolderBase_Position);
pByte[1]	:= DINT_TO_BYTE(VariantsBroachingPlan.ToolHolderA_Position);
pByte[2]	:= DINT_TO_BYTE(VariantsBroachingPlan.ToolHolderB_Position);
pByte[3]	:= DINT_TO_BYTE(VariantsBroachingPlan.ToolHolderC_Position);
pByte[4]	:= DINT_TO_BYTE(VariantsBroachingPlan.ToolHolderD_Position);
pByte[5] 	:= DINT_TO_BYTE(VariantsBroachingPlan.ToolHolderE_Position);
pByte[6] 	:= DINT_TO_BYTE(VariantsBroachingPlan.ToolHolderF_Position);

END_FUNCTION

// ---- FBs/DataRequest/FC_BroachingPlanCopyConpensation.TcPOU
FUNCTION FC_BroachingPlanCopyConpensation
VAR_INPUT
	pDWord : POINTER TO DWORD;
	BaseBroachingPlan 		: DUT_stBroachingPlanBase;     
    VariantsBroachingPlan	: DUT_stBroachingPlanVariants;
END_VAR

			// correzioni master 
			pDWord[0] := REAL_TO_DWORD(BaseBroachingPlan.ToolHolderBase_AngleCompensation * 1000.0);
			pDWord[1] := REAL_TO_DWORD(BaseBroachingPlan.ToolHolderBase_LateralCompensation * 1000.0);
			pDWord[2] := REAL_TO_DWORD(BaseBroachingPlan.ToolHolderBase_DepthCompensation * 1000.0);
			
			// correzioni variante 1 
			pDWord[3] := REAL_TO_DWORD(VariantsBroachingPlan.ToolHolderA_AngleCompensation * 1000.0);
			pDWord[4] := REAL_TO_DWORD(VariantsBroachingPlan.ToolHolderA_LateralCompensation * 1000.0);
			pDWord[5] := REAL_TO_DWORD(VariantsBroachingPlan.ToolHolderA_DepthCompensation * 1000.0);			
			
			// correzioni variante 2 
			pDWord[6] := REAL_TO_DWORD(VariantsBroachingPlan.ToolHolderB_AngleCompensation * 1000.0);
			pDWord[7] := REAL_TO_DWORD(VariantsBroachingPlan.ToolHolderB_LateralCompensation * 1000.0);
			pDWord[8] := REAL_TO_DWORD(VariantsBroachingPlan.ToolHolderB_DepthCompensation * 1000.0);			
			
			// correzioni variante 3 
			pDWord[9] := REAL_TO_DWORD(VariantsBroachingPlan.ToolHolderC_AngleCompensation * 1000.0);
			pDWord[10] := REAL_TO_DWORD(VariantsBroachingPlan.ToolHolderC_LateralCompensation * 1000.0);
			pDWord[11] := REAL_TO_DWORD(VariantsBroachingPlan.ToolHolderC_DepthCompensation * 1000.0);			
			
			// correzioni variante 4 
			pDWord[12] := REAL_TO_DWORD(VariantsBroachingPlan.ToolHolderD_AngleCompensation * 1000.0);
			pDWord[13] := REAL_TO_DWORD(VariantsBroachingPlan.ToolHolderD_LateralCompensation * 1000.0);
			pDWord[14] := REAL_TO_DWORD(VariantsBroachingPlan.ToolHolderD_DepthCompensation * 1000.0);			
			
			// correzioni variante 5 
			pDWord[15] := REAL_TO_DWORD(VariantsBroachingPlan.ToolHolderE_AngleCompensation * 1000.0);
			pDWord[16] := REAL_TO_DWORD(VariantsBroachingPlan.ToolHolderE_LateralCompensation * 1000.0);
			pDWord[17] := REAL_TO_DWORD(VariantsBroachingPlan.ToolHolderE_DepthCompensation * 1000.0);			
			
			// correzioni variante 6 
			pDWord[18] := REAL_TO_DWORD(VariantsBroachingPlan.ToolHolderF_AngleCompensation * 1000.0);
			pDWord[19] := REAL_TO_DWORD(VariantsBroachingPlan.ToolHolderF_LateralCompensation * 1000.0);
			pDWord[20] := REAL_TO_DWORD(VariantsBroachingPlan.ToolHolderF_DepthCompensation * 1000.0);

END_FUNCTION

// ---- FBs/FB_OvrMng.TcPOU
FUNCTION_BLOCK FB_OvrMng
// Funzione per la gestione della scheda encoder EP5151 utilizzata per la lettura del potenziometro di override
// Sotto è riportata la configurazione della scheda EP5151
VAR_INPUT
	I_CounterValue       : UINT;    // Valore attuale del contatore encoder
    I_SetCounterDone     : BOOL;    // Stato dell'operazione di set del contatore (TRUE se avvenuta con successo)
    I_Overflow           : BOOL;    // Segnalazione di overflow del contatore
    I_Underflow          : BOOL;    // Segnalazione di underflow del contatore
    I_Multiplier         : USINT;   // Moltiplicatore per incrementi del potenziometro di override
    I_SetCounter         : BOOL;    // Comando per il set manuale del contatore
    I_SetCounterValue    : UINT;    // Valore da impostare nel contatore tramite comando di set
    I_OvrMaxValue        : USINT;   // Limite massimo per il valore di override
    I_OvrMinValue        : USINT;   // Limite minimo per il valore di override
END_VAR                  
VAR_OUTPUT               
	Q_SetCounter        : BOOL;     // Stato del comando di set del contatore (attivo quando il contatore è impostato)
    Q_SetCounterValue   : UINT;     // Valore al quale il contatore è impostato quando il comando di set è attivo
END_VAR
VAR_IN_OUT
    I_CounterValueOld   : UINT;     // Valore precedente del contatore, usato per rilevare variazioni (variabile retentiva)
    Q_Ovr               : USINT;    // Valore di override limitato ai valori massimo e minimo
END_VAR
VAR
	diff					: DINT;
	OvrTemp					: DINT;
	RTRIG_SetCounter		: R_TRIG;
END_VAR
//8000:0     ENC Settings                     RW       > 23 <
//8000:01    Enable C reset                   RW       FALSE
//8000:02    Enable extern reset              RW       FALSE
//8000:03    Enable up/down counter           RW       TRUE
//8000:04    Gate polarity                    RW       Enable pos. gate (1)
//8000:08    Disable filter                   RW       FALSE
//8000:0A    Enable micro increments          RW       FALSE
//8000:0B    Open circuit detection A         RW       TRUE
//8000:0C    Open circuit detection B         RW       TRUE
//8000:0D    Open circuit detection C         RW       TRUE
//8000:0E    Reversion of rotation            RW       FALSE
//8000:10    Extern reset polarity            RW       Rise (1)
//8000:11    Frequency window                 RW       0x2710 (10000)
//8000:13    Frequency scaling                RW       0.01Hz (100)
//8000:14    Period scaling                   RW       100ns (100)
//8000:15    Frequency resolution             RW       0.01Hz (100)
//8000:16    Period resolution                RW       100ns (100)
//8000:17    Frequency wait time              RW       0x0640 (1600)

// Inizializza il valore dell'override con il valore salvato nella variabile retentiva
OvrTemp := Q_Ovr;

// Aggiorna il valore del contatore dopo una variazione
IF I_CounterValueOld <> I_CounterValue AND NOT Q_SetCounter THEN
	diff := I_CounterValue - I_CounterValueOld;

 // Gestisce overflow e underflow del contatore	
	IF diff > 32767 THEN
		diff := diff - 65536;
	ELSIF diff < -32768 THEN 
		diff := diff + 65536;
	END_IF

// Gestisce variazioni doppie causate da un singolo click della manopola (purtroppo la scheda si comporta in questo modo)
// 1 click della manopola corrisponde a una variazione di ±2
	IF ABS(diff) > 1 THEN
		I_CounterValueOld := I_CounterValue;
		OvrTemp := OvrTemp + (diff*I_Multiplier)/2;

// Gestisce overflow e underflow a livello di scheda
// Se si verifica un overflow o underflow, forza il contatore al valore massimo/2 per evitare condizioni di overflow persistenti
		IF I_Overflow OR I_Underflow  AND NOT Q_SetCounter THEN
			SetCounter(32767);
		END_IF
	END_IF
END_IF

// Gestione del set manuale del contatore; consente il controllo esterno del conteggio
RTRIG_SetCounter(CLK := I_SetCounter);
IF RTRIG_SetCounter.Q AND NOT Q_SetCounter THEN
	SetCounter(I_SetCounterValue);
END_IF
IF Q_SetCounter AND I_SetCounterDone THEN
	Q_SetCounter := FALSE;
END_IF
//////

// Limita e applica il valore di override, rispettando i limiti massimo e minimo
Q_Ovr := SEL(
	OvrTemp > I_OvrMaxValue, 
	(SEL(OvrTemp < I_OvrMinValue, (DINT_TO_USINT(OvrTemp)), I_OvrMinValue)), 
	I_OvrMaxValue
);

METHOD SetCounter : BOOL
VAR_INPUT
	CounterValue : UINT; // valore a cui forzare il conteggio
END_VAR
Q_SetCounterValue := I_CounterValueOld := CounterValue;
Q_SetCounter := TRUE;
END_METHOD

END_FUNCTION_BLOCK

// ---- FBs/FB_ButtonTrigger.TcPOU
FUNCTION_BLOCK FB_ButtonTrigger
VAR_INPUT
	I_Command		: BOOL;
	I_CommandEnable	: BOOL;
	I_Reset			: BOOL;
	I_ResetEnable	: BOOL;
END_VAR
VAR_IN_OUT
	Q_Out			: BOOL;
END_VAR
VAR
	RTRIG_Set	: R_TRIG;
	RTRIG_Reset	: R_TRIG;
END_VAR

RTRIG_Set(CLK := I_Command);
RTRIG_Reset(CLK := I_Reset);

IF RTRIG_Reset.Q AND I_ResetEnable THEN
	Q_Out := FALSE;
ELSIF RTRIG_Set.Q AND I_CommandEnable THEN
	Q_Out := TRUE;
END_IF

END_FUNCTION_BLOCK

// ---- FBs/FB_LoadingModeChange.TcPOU
FUNCTION_BLOCK FB_LoadingModeChange
VAR_INPUT
	LoadingModeSelected : eLoadingMode;	
	LS_AutoMode		: BOOL;
	LS_ManualMode	: BOOL;
	LS_SemiAutoMode : BOOL; 
END_VAR
VAR_OUTPUT
	PS_AutoMode		: BOOL;
	PS_ManualMode	: BOOL;
	PS_SemiAutoMode : BOOL;
END_VAR
VAR_IN_OUT
	ActualMode : eLoadingMode;
END_VAR
VAR
	RTRIG_AutoMode :  R_TRIG;
	RTRIG_ManualMode :  R_TRIG;
	RTRIG_SemiAutoMode :  R_TRIG;
END_VAR

RTRIG_AutoMode(CLK := LS_AutoMode);
RTRIG_ManualMode(CLK := LS_ManualMode);
RTRIG_SemiAutoMode(CLK := LS_SemiAutoMode);

//IF LoadingModeSelected <> ActualMode THEN
	IF LoadingModeSelected = eLoadingMOde.Auto THEN
		PS_AutoMode := TRUE;
		PS_ManualMode := FALSE;
		PS_SemiAutoMOde := FALSE;
	ELSIF LoadingModeSelected = eLoadingMOde.Manual THEN
		PS_AutoMode := FALSE;
		PS_ManualMode := TRUE;
		PS_SemiAutoMOde := FALSE;
	ELSIF LoadingModeSelected = eLoadingMOde.SemiAuto THEN
		PS_AutoMode := FALSE;
		PS_ManualMode := FALSE;
		PS_SemiAutoMOde := TRUE;
	ELSE
		PS_AutoMode := FALSE;
		PS_ManualMode := FALSE;
		PS_SemiAutoMOde := FALSE;		
	END_IF
//END_IF

IF RTRIG_AutoMode.Q THEN
	PS_AutoMode := FALSE;
	PS_ManualMode := FALSE;
	PS_SemiAutoMOde := FALSE;
	ActualMode := eLoadingMode.Auto;	
END_IF

IF RTRIG_ManualMode.Q THEN
	PS_AutoMode := FALSE;
	PS_ManualMode := FALSE;
	PS_SemiAutoMOde := FALSE;
	ActualMode := eLoadingMode.Manual;	
END_IF

IF RTRIG_SemiAutoMode.Q THEN
	PS_AutoMode := FALSE;
	PS_ManualMode := FALSE;
	PS_SemiAutoMOde := FALSE;
	ActualMode := eLoadingMode.SemiAuto;	
END_IF

END_FUNCTION_BLOCK

// ---- FBs/FB_KillMultipleNavigationPS.TcPOU
FUNCTION_BLOCK FB_KillMultipleNavigationPS
VAR_INPUT
	Ps	: POINTER TO BOOL;
END_VAR
VAR
	i : USINT;
	activeCount : UINT;
	TON_DelayResetPs : TON;
END_VAR

activeCount := 0;
FOR i := 0 TO 20 DO
    IF Ps[i] THEN
        activeCount := activeCount + 1;
    END_IF
END_FOR

TON_DelayResetPs(IN := activeCount > 1, PT := T#500MS);

IF TON_DelayResetPs.Q THEN
	MEMSET(Ps, 0, SIZEOF(HMI.In.Navigation.PS)-SIZEOF(BOOL));
	activeCount := 0;
END_IF

END_FUNCTION_BLOCK

// ---- POUs/PRG_Diagnostic.TcPOU
PROGRAM PRG_Diagnostic
VAR
	i: UDINT;
	StAlr	 : ARRAY[0..CNC.NUM_STATIONS+4] OF ARRAY[0..CNC.NUM_MAX_STATION_ALARMS-1] OF BOOL;
	fbEVSt00 : ARRAY[0..CNC.NUM_MAX_MANUALS_00-1] OF FB_PneumaticActuator_2EV_Diagnostic;
	fbEVSt01 : ARRAY[0..CNC.NUM_MAX_MANUALS_01-1] OF FB_PneumaticActuator_2EV_Diagnostic;
	fbEVSt02 : ARRAY[0..CNC.NUM_MAX_MANUALS_02-1] OF FB_PneumaticActuator_2EV_Diagnostic;
	fbEVSt03 : ARRAY[0..CNC.NUM_MAX_MANUALS_03-1] OF FB_PneumaticActuator_2EV_Diagnostic;
	fbEVSt04 : ARRAY[0..CNC.NUM_MAX_MANUALS_04-1] OF FB_PneumaticActuator_2EV_Diagnostic;
	fbEVSt05 : ARRAY[0..CNC.NUM_MAX_MANUALS_05-1] OF FB_PneumaticActuator_2EV_Diagnostic;
	fbEVSt06 : ARRAY[0..CNC.NUM_MAX_MANUALS_06-1] OF FB_PneumaticActuator_2EV_Diagnostic;
	fbEVSt07 : ARRAY[0..CNC.NUM_MAX_MANUALS_07-1] OF FB_PneumaticActuator_2EV_Diagnostic;
	fbEVSt08 : ARRAY[0..CNC.NUM_MAX_MANUALS_08-1] OF FB_PneumaticActuator_2EV_Diagnostic;
	fbEVSt09 : ARRAY[0..CNC.NUM_MAX_MANUALS_09-1] OF FB_PneumaticActuator_2EV_Diagnostic;
	fbEVSt10 : ARRAY[0..CNC.NUM_MAX_MANUALS_10-1] OF FB_PneumaticActuator_2EV_Diagnostic;
	fbEVSt11 : ARRAY[0..CNC.NUM_MAX_MANUALS_11-1] OF FB_PneumaticActuator_2EV_Diagnostic;
	fbEVSt12 : ARRAY[0..CNC.NUM_MAX_MANUALS_12-1] OF FB_PneumaticActuator_2EV_Diagnostic;
	fbEVSt13 : ARRAY[0..CNC.NUM_MAX_MANUALS_13-1] OF FB_PneumaticActuator_2EV_Diagnostic;	
END_VAR

A_01_EVDiagnostic();
A_02_EVDiagnostic();
A_03_EVDiagnostic();
A_04_EVDiagnostic();
A_05_EVDiagnostic();
A_06_EVDiagnostic();
A_07_EVDiagnostic();
A_08_EVDiagnostic();
A_09_EVDiagnostic();
A_10_EVDiagnostic();
A_11_EVDiagnostic();
A_12_EVDiagnostic();
A_13_EVDiagnostic();

A_01_Alarms();

ACTION A_00_Alarms:
FOR i:= 0 TO CNC.NUM_MAX_STATION_ALARMS -1 DO 
	StAlr[0][i] := PRG_EventManagement._PMCEventCollectors._CheckFanucPMCActiveAlarmList_St00_Alr._PMCEvents[i].bRaised;
END_FOR

HMI.St0.EVInfo[64].Error := PRG_Diagnostic.fbEVSt00[0].Q_eStatus = eEV_Status.MovingForward AND StAlr[1][0];		
HMI.St0.EVInfo[65].Error := PRG_Diagnostic.fbEVSt00[0].Q_eStatus = eEV_Status.MovingBackward AND StAlr[1][0];
HMI.St0.EVInfo[64].Error := PRG_Diagnostic.fbEVSt00[1].Q_eStatus = eEV_Status.MovingForward AND StAlr[1][0];
HMI.St0.EVInfo[65].Error := PRG_Diagnostic.fbEVSt00[1].Q_eStatus = eEV_Status.MovingBackward AND StAlr[1][0]; 
      
HMI.St0.EVInfo[66].dTime := PRG_Diagnostic.fbEVSt00[0].Q_tElapsedTimeFwd;		
HMI.St0.EVInfo[67].dTime := PRG_Diagnostic.fbEVSt00[0].Q_tElapsedTimeBwd;
HMI.St0.EVInfo[66].dTime := PRG_Diagnostic.fbEVSt00[1].Q_tElapsedTimeFwd;
HMI.St0.EVInfo[67].dTime := PRG_Diagnostic.fbEVSt00[1].Q_tElapsedTimeBwd;
END_ACTION

ACTION A_00_EVDiagnostic:
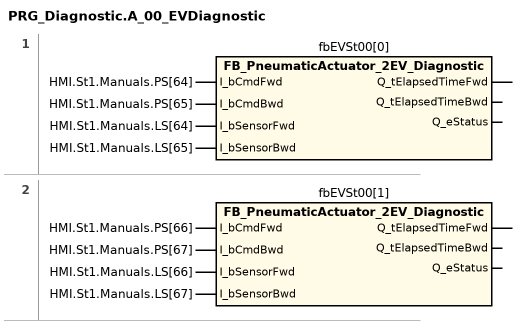
// NETWORK 1
fbEVSt00[0](
    I_bCmdFwd := HMI.St1.Manuals.PS[64],
    I_bCmdBwd := HMI.St1.Manuals.PS[65],
    I_bSensorFwd := HMI.St1.Manuals.LS[64],
    I_bSensorBwd := HMI.St1.Manuals.LS[65]); // FB_PneumaticActuator_2EV_Diagnostic

// NETWORK 2
fbEVSt00[1](
    I_bCmdFwd := HMI.St1.Manuals.PS[66],
    I_bCmdBwd := HMI.St1.Manuals.PS[67],
    I_bSensorFwd := HMI.St1.Manuals.LS[66],
    I_bSensorBwd := HMI.St1.Manuals.LS[67]); // FB_PneumaticActuator_2EV_Diagnostic
END_ACTION

ACTION A_01_Alarms:
FOR i:= 0 TO CNC.NUM_MAX_STATION_ALARMS -1 DO 
	StAlr[1][i] := PRG_EventManagement._PMCEventCollectors._CheckFanucPMCActiveAlarmList_St01_Alr._PMCEvents[i].bRaised;
END_FOR

HMI.St1.EVInfo[32].Error := PRG_Diagnostic.fbEVSt01[0].Q_eStatus = eEV_Status.MovingForward AND StAlr[1][0];		
HMI.St1.EVInfo[33].Error := PRG_Diagnostic.fbEVSt01[0].Q_eStatus = eEV_Status.MovingBackward AND StAlr[1][0];
HMI.St1.EVInfo[34].Error := PRG_Diagnostic.fbEVSt01[1].Q_eStatus = eEV_Status.MovingForward AND StAlr[1][0];
HMI.St1.EVInfo[35].Error := PRG_Diagnostic.fbEVSt01[1].Q_eStatus = eEV_Status.MovingBackward AND StAlr[1][0]; 
HMI.St1.EVInfo[36].Error := PRG_Diagnostic.fbEVSt01[2].Q_eStatus = eEV_Status.MovingForward AND StAlr[1][0];		
HMI.St1.EVInfo[37].Error := PRG_Diagnostic.fbEVSt01[2].Q_eStatus = eEV_Status.MovingBackward AND StAlr[1][0]; 
HMI.St1.EVInfo[25].Error := PRG_Diagnostic.fbEVSt01[3].Q_eStatus = eEV_Status.MovingForward AND StAlr[1][0];		
HMI.St1.EVInfo[26].Error := PRG_Diagnostic.fbEVSt01[3].Q_eStatus = eEV_Status.MovingBackward AND StAlr[1][0]; 

HMI.St1.EVInfo[32].dTime := PRG_Diagnostic.fbEVSt01[0].Q_tElapsedTimeFwd;		
HMI.St1.EVInfo[33].dTime := PRG_Diagnostic.fbEVSt01[0].Q_tElapsedTimeBwd;
HMI.St1.EVInfo[34].dTime := PRG_Diagnostic.fbEVSt01[1].Q_tElapsedTimeFwd;
HMI.St1.EVInfo[35].dTime := PRG_Diagnostic.fbEVSt01[1].Q_tElapsedTimeBwd;
HMI.St1.EVInfo[36].dTime := PRG_Diagnostic.fbEVSt01[2].Q_tElapsedTimeFwd;		
HMI.St1.EVInfo[37].dTime := PRG_Diagnostic.fbEVSt01[2].Q_tElapsedTimeBwd;
HMI.St1.EVInfo[25].dTime := PRG_Diagnostic.fbEVSt01[3].Q_tElapsedTimeFwd;		
HMI.St1.EVInfo[26].dTime := PRG_Diagnostic.fbEVSt01[3].Q_tElapsedTimeBwd;
END_ACTION

ACTION A_01_EVDiagnostic:
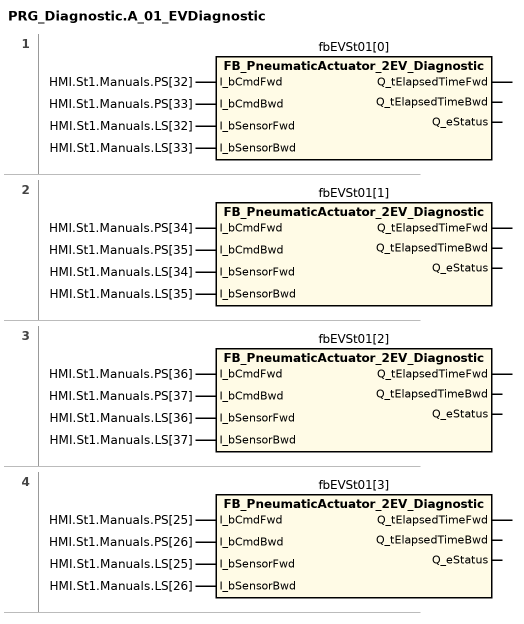
// NETWORK 1
fbEVSt01[0](
    I_bCmdFwd := HMI.St1.Manuals.PS[32],
    I_bCmdBwd := HMI.St1.Manuals.PS[33],
    I_bSensorFwd := HMI.St1.Manuals.LS[32],
    I_bSensorBwd := HMI.St1.Manuals.LS[33]); // FB_PneumaticActuator_2EV_Diagnostic

// NETWORK 2
fbEVSt01[1](
    I_bCmdFwd := HMI.St1.Manuals.PS[34],
    I_bCmdBwd := HMI.St1.Manuals.PS[35],
    I_bSensorFwd := HMI.St1.Manuals.LS[34],
    I_bSensorBwd := HMI.St1.Manuals.LS[35]); // FB_PneumaticActuator_2EV_Diagnostic

// NETWORK 3
fbEVSt01[2](
    I_bCmdFwd := HMI.St1.Manuals.PS[36],
    I_bCmdBwd := HMI.St1.Manuals.PS[37],
    I_bSensorFwd := HMI.St1.Manuals.LS[36],
    I_bSensorBwd := HMI.St1.Manuals.LS[37]); // FB_PneumaticActuator_2EV_Diagnostic

// NETWORK 4
fbEVSt01[3](
    I_bCmdFwd := HMI.St1.Manuals.PS[25],
    I_bCmdBwd := HMI.St1.Manuals.PS[26],
    I_bSensorFwd := HMI.St1.Manuals.LS[25],
    I_bSensorBwd := HMI.St1.Manuals.LS[26]); // FB_PneumaticActuator_2EV_Diagnostic
END_ACTION

ACTION A_02_Alarms:
FOR i:= 0 TO CNC.NUM_MAX_STATION_ALARMS -1 DO 
	StAlr[2][i] := PRG_EventManagement._PMCEventCollectors._CheckFanucPMCActiveAlarmList_St02_Alr._PMCEvents[i].bRaised;
END_FOR

HMI.St2.EVInfo[32].Error := PRG_Diagnostic.fbEVSt02[0].Q_eStatus = eEV_Status.MovingForward  AND StAlr[2][0];		
HMI.St2.EVInfo[33].Error := PRG_Diagnostic.fbEVSt02[0].Q_eStatus = eEV_Status.MovingBackward AND StAlr[2][0];
HMI.St2.EVInfo[34].Error := PRG_Diagnostic.fbEVSt02[1].Q_eStatus = eEV_Status.MovingForward  AND StAlr[2][0];
HMI.St2.EVInfo[35].Error := PRG_Diagnostic.fbEVSt02[1].Q_eStatus = eEV_Status.MovingBackward AND StAlr[2][0]; 
                                                  
HMI.St2.EVInfo[32].dTime := PRG_Diagnostic.fbEVSt02[0].Q_tElapsedTimeFwd;		
HMI.St2.EVInfo[33].dTime := PRG_Diagnostic.fbEVSt02[0].Q_tElapsedTimeBwd;
HMI.St2.EVInfo[34].dTime := PRG_Diagnostic.fbEVSt02[1].Q_tElapsedTimeFwd;
HMI.St2.EVInfo[35].dTime := PRG_Diagnostic.fbEVSt02[1].Q_tElapsedTimeBwd;
END_ACTION

ACTION A_02_EVDiagnostic:
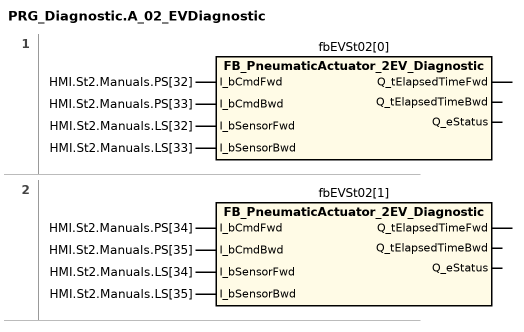
// NETWORK 1
fbEVSt02[0](
    I_bCmdFwd := HMI.St2.Manuals.PS[32],
    I_bCmdBwd := HMI.St2.Manuals.PS[33],
    I_bSensorFwd := HMI.St2.Manuals.LS[32],
    I_bSensorBwd := HMI.St2.Manuals.LS[33]); // FB_PneumaticActuator_2EV_Diagnostic

// NETWORK 2
fbEVSt02[1](
    I_bCmdFwd := HMI.St2.Manuals.PS[34],
    I_bCmdBwd := HMI.St2.Manuals.PS[35],
    I_bSensorFwd := HMI.St2.Manuals.LS[34],
    I_bSensorBwd := HMI.St2.Manuals.LS[35]); // FB_PneumaticActuator_2EV_Diagnostic
END_ACTION

ACTION A_03_Alarms:
FOR i:= 0 TO CNC.NUM_MAX_STATION_ALARMS -1 DO 
	StAlr[3][i] := PRG_EventManagement._PMCEventCollectors._CheckFanucPMCActiveAlarmList_St03_Alr._PMCEvents[i].bRaised;
END_FOR

HMI.St3.EVInfo[33].Error := PRG_Diagnostic.fbEVSt03[0].Q_eStatus = eEV_Status.MovingForward  AND StAlr[3][0];		
HMI.St3.EVInfo[32].Error := PRG_Diagnostic.fbEVSt03[0].Q_eStatus = eEV_Status.MovingBackward AND StAlr[3][0];
      
HMI.St3.EVInfo[33].dTime := PRG_Diagnostic.fbEVSt03[0].Q_tElapsedTimeFwd;		
HMI.St3.EVInfo[32].dTime := PRG_Diagnostic.fbEVSt03[0].Q_tElapsedTimeBwd;
END_ACTION

ACTION A_03_EVDiagnostic:
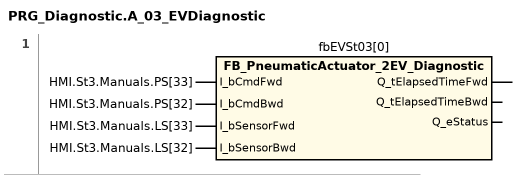
// NETWORK 1
fbEVSt03[0](
    I_bCmdFwd := HMI.St3.Manuals.PS[33],
    I_bCmdBwd := HMI.St3.Manuals.PS[32],
    I_bSensorFwd := HMI.St3.Manuals.LS[33],
    I_bSensorBwd := HMI.St3.Manuals.LS[32]); // FB_PneumaticActuator_2EV_Diagnostic
END_ACTION

ACTION A_04_Alarms:
FOR i:= 0 TO CNC.NUM_MAX_STATION_ALARMS -1 DO 
	StAlr[4][i] := PRG_EventManagement._PMCEventCollectors._CheckFanucPMCActiveAlarmList_St04_Alr._PMCEvents[i].bRaised;
END_FOR

HMI.St4.EVInfo[36].Error := PRG_Diagnostic.fbEVSt04[2].Q_eStatus = eEV_Status.MovingForward  AND StAlr[4][0];
HMI.St4.EVInfo[37].Error := PRG_Diagnostic.fbEVSt04[2].Q_eStatus = eEV_Status.MovingBackward AND StAlr[4][0]; 
HMI.St4.EVInfo[38].Error := PRG_Diagnostic.fbEVSt04[3].Q_eStatus = eEV_Status.MovingForward  AND StAlr[4][0];		
HMI.St4.EVInfo[39].Error := PRG_Diagnostic.fbEVSt04[3].Q_eStatus = eEV_Status.MovingBackward AND StAlr[4][0]; 
                                                  
HMI.St4.EVInfo[36].dTime := PRG_Diagnostic.fbEVSt04[2].Q_tElapsedTimeFwd;		
HMI.St4.EVInfo[37].dTime := PRG_Diagnostic.fbEVSt04[2].Q_tElapsedTimeBwd;
HMI.St4.EVInfo[38].dTime := PRG_Diagnostic.fbEVSt04[3].Q_tElapsedTimeFwd;
HMI.St4.EVInfo[39].dTime := PRG_Diagnostic.fbEVSt04[3].Q_tElapsedTimeBwd;
END_ACTION

ACTION A_04_EVDiagnostic:
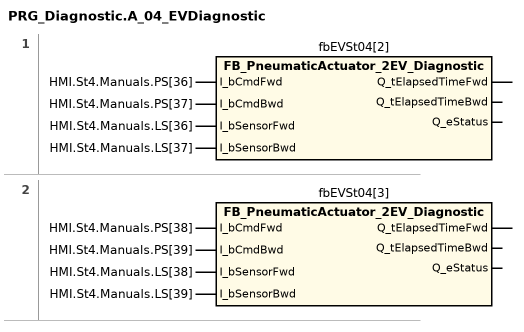
// NETWORK 1
fbEVSt04[2](
    I_bCmdFwd := HMI.St4.Manuals.PS[36],
    I_bCmdBwd := HMI.St4.Manuals.PS[37],
    I_bSensorFwd := HMI.St4.Manuals.LS[36],
    I_bSensorBwd := HMI.St4.Manuals.LS[37]); // FB_PneumaticActuator_2EV_Diagnostic

// NETWORK 2
fbEVSt04[3](
    I_bCmdFwd := HMI.St4.Manuals.PS[38],
    I_bCmdBwd := HMI.St4.Manuals.PS[39],
    I_bSensorFwd := HMI.St4.Manuals.LS[38],
    I_bSensorBwd := HMI.St4.Manuals.LS[39]); // FB_PneumaticActuator_2EV_Diagnostic
END_ACTION

ACTION A_05_Alarms:
FOR i:= 0 TO CNC.NUM_MAX_STATION_ALARMS -1 DO 
	StAlr[5][i] := PRG_EventManagement._PMCEventCollectors._CheckFanucPMCActiveAlarmList_St05_Alr._PMCEvents[i].bRaised;
END_FOR

HMI.St5.EVInfo[40].Error := PRG_Diagnostic.fbEVSt05[4].Q_eStatus  = eEV_Status.MovingForward  AND StAlr[5][0];		
HMI.St5.EVInfo[41].Error := PRG_Diagnostic.fbEVSt05[4].Q_eStatus  = eEV_Status.MovingBackward AND StAlr[5][0];
HMI.St5.EVInfo[64].Error := PRG_Diagnostic.fbEVSt05[16].Q_eStatus = eEV_Status.MovingForward  AND StAlr[5][0];
HMI.St5.EVInfo[65].Error := PRG_Diagnostic.fbEVSt05[16].Q_eStatus = eEV_Status.MovingBackward AND StAlr[5][0]; 
HMI.St5.EVInfo[66].Error := PRG_Diagnostic.fbEVSt05[17].Q_eStatus = eEV_Status.MovingForward  AND StAlr[5][0];		
HMI.St5.EVInfo[67].Error := PRG_Diagnostic.fbEVSt05[17].Q_eStatus = eEV_Status.MovingBackward AND StAlr[5][0]; 
                                                  
HMI.St5.EVInfo[40].dTime := PRG_Diagnostic.fbEVSt05[4].Q_tElapsedTimeFwd;		
HMI.St5.EVInfo[41].dTime := PRG_Diagnostic.fbEVSt05[4].Q_tElapsedTimeBwd;
HMI.St5.EVInfo[64].dTime := PRG_Diagnostic.fbEVSt05[16].Q_tElapsedTimeFwd;
HMI.St5.EVInfo[65].dTime := PRG_Diagnostic.fbEVSt05[16].Q_tElapsedTimeBwd;
HMI.St5.EVInfo[66].dTime := PRG_Diagnostic.fbEVSt05[17].Q_tElapsedTimeFwd;		
HMI.St5.EVInfo[67].dTime := PRG_Diagnostic.fbEVSt05[17].Q_tElapsedTimeBwd;
END_ACTION

ACTION A_05_EVDiagnostic:
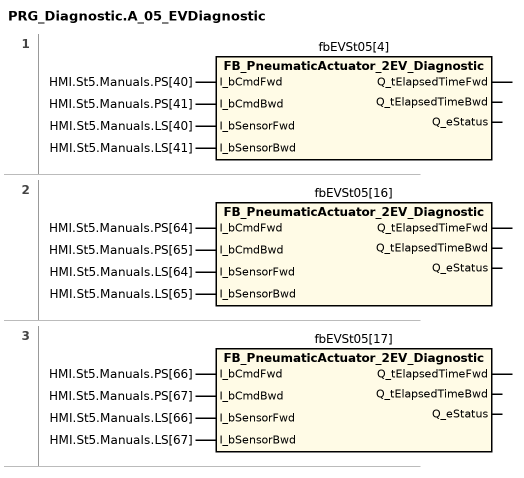
// NETWORK 1
fbEVSt05[4](
    I_bCmdFwd := HMI.St5.Manuals.PS[40],
    I_bCmdBwd := HMI.St5.Manuals.PS[41],
    I_bSensorFwd := HMI.St5.Manuals.LS[40],
    I_bSensorBwd := HMI.St5.Manuals.LS[41]); // FB_PneumaticActuator_2EV_Diagnostic

// NETWORK 2
fbEVSt05[16](
    I_bCmdFwd := HMI.St5.Manuals.PS[64],
    I_bCmdBwd := HMI.St5.Manuals.PS[65],
    I_bSensorFwd := HMI.St5.Manuals.LS[64],
    I_bSensorBwd := HMI.St5.Manuals.LS[65]); // FB_PneumaticActuator_2EV_Diagnostic

// NETWORK 3
fbEVSt05[17](
    I_bCmdFwd := HMI.St5.Manuals.PS[66],
    I_bCmdBwd := HMI.St5.Manuals.PS[67],
    I_bSensorFwd := HMI.St5.Manuals.LS[66],
    I_bSensorBwd := HMI.St5.Manuals.LS[67]); // FB_PneumaticActuator_2EV_Diagnostic
END_ACTION

ACTION A_06_Alarms:
FOR i:= 0 TO CNC.NUM_MAX_STATION_ALARMS -1 DO 
	StAlr[6][i] := PRG_EventManagement._PMCEventCollectors._CheckFanucPMCActiveAlarmList_St06_Alr._PMCEvents[i].bRaised;
END_FOR

HMI.St6.EVInfo[40].Error := PRG_Diagnostic.fbEVSt06[4].Q_eStatus = eEV_Status.MovingForward  AND StAlr[6][0];		
HMI.St6.EVInfo[41].Error := PRG_Diagnostic.fbEVSt06[4].Q_eStatus = eEV_Status.MovingBackward AND StAlr[6][0]; 

HMI.St6.EVInfo[40].dTime := PRG_Diagnostic.fbEVSt06[4].Q_tElapsedTimeFwd;		
HMI.St6.EVInfo[41].dTime := PRG_Diagnostic.fbEVSt06[4].Q_tElapsedTimeBwd;
END_ACTION

ACTION A_06_EVDiagnostic:
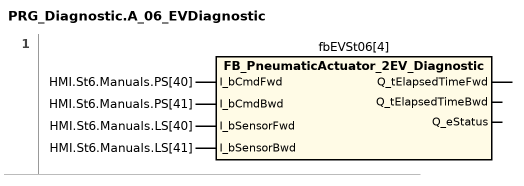
// NETWORK 1
fbEVSt06[4](
    I_bCmdFwd := HMI.St6.Manuals.PS[40],
    I_bCmdBwd := HMI.St6.Manuals.PS[41],
    I_bSensorFwd := HMI.St6.Manuals.LS[40],
    I_bSensorBwd := HMI.St6.Manuals.LS[41]); // FB_PneumaticActuator_2EV_Diagnostic
END_ACTION

ACTION A_07_Alarms:
FOR i:= 0 TO CNC.NUM_MAX_STATION_ALARMS -1 DO 
	StAlr[7][i] := PRG_EventManagement._PMCEventCollectors._CheckFanucPMCActiveAlarmList_St07_Alr._PMCEvents[i].bRaised;
END_FOR

HMI.St1.EVInfo[40].Error := PRG_Diagnostic.fbEVSt07[4].Q_eStatus = eEV_Status.MovingForward  AND StAlr[7][0];		
HMI.St1.EVInfo[41].Error := PRG_Diagnostic.fbEVSt07[4].Q_eStatus = eEV_Status.MovingBackward AND StAlr[7][0];

HMI.St1.EVInfo[40].dTime := PRG_Diagnostic.fbEVSt07[4].Q_tElapsedTimeFwd;		
HMI.St1.EVInfo[41].dTime := PRG_Diagnostic.fbEVSt07[4].Q_tElapsedTimeBwd;
END_ACTION

ACTION A_07_EVDiagnostic:
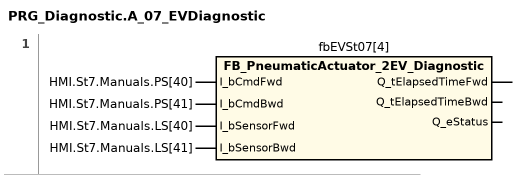
// NETWORK 1
fbEVSt07[4](
    I_bCmdFwd := HMI.St7.Manuals.PS[40],
    I_bCmdBwd := HMI.St7.Manuals.PS[41],
    I_bSensorFwd := HMI.St7.Manuals.LS[40],
    I_bSensorBwd := HMI.St7.Manuals.LS[41]); // FB_PneumaticActuator_2EV_Diagnostic
END_ACTION

ACTION A_08_Alarms:
FOR i:= 0 TO CNC.NUM_MAX_STATION_ALARMS -1 DO 
	StAlr[8][i] := PRG_EventManagement._PMCEventCollectors._CheckFanucPMCActiveAlarmList_St08_Alr._PMCEvents[i].bRaised;
END_FOR

HMI.St8.EVInfo[40].Error := PRG_Diagnostic.fbEVSt08[0].Q_eStatus = eEV_Status.MovingForward  AND StAlr[8][0];		
HMI.St8.EVInfo[41].Error := PRG_Diagnostic.fbEVSt08[0].Q_eStatus = eEV_Status.MovingBackward AND StAlr[8][0];

HMI.St8.EVInfo[40].dTime := PRG_Diagnostic.fbEVSt08[0].Q_tElapsedTimeFwd;		
HMI.St8.EVInfo[41].dTime := PRG_Diagnostic.fbEVSt08[0].Q_tElapsedTimeBwd;
END_ACTION

ACTION A_08_EVDiagnostic:
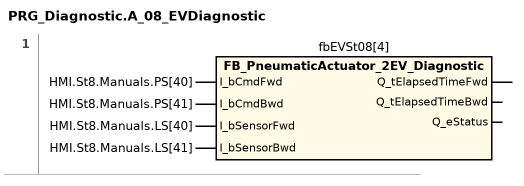
// NETWORK 1
fbEVSt08[4](
    I_bCmdFwd := HMI.St8.Manuals.PS[40],
    I_bCmdBwd := HMI.St8.Manuals.PS[41],
    I_bSensorFwd := HMI.St8.Manuals.LS[40],
    I_bSensorBwd := HMI.St8.Manuals.LS[41]); // FB_PneumaticActuator_2EV_Diagnostic
END_ACTION

ACTION A_09_Alarms:
FOR i:= 0 TO CNC.NUM_MAX_STATION_ALARMS -1 DO 
	StAlr[9][i] := PRG_EventManagement._PMCEventCollectors._CheckFanucPMCActiveAlarmList_St09_Alr._PMCEvents[i].bRaised;
END_FOR

HMI.St9.EVInfo[40].Error := PRG_Diagnostic.fbEVSt09[4].Q_eStatus = eEV_Status.MovingForward  AND StAlr[1][0];		
HMI.St9.EVInfo[41].Error := PRG_Diagnostic.fbEVSt09[4].Q_eStatus = eEV_Status.MovingBackward AND StAlr[1][0];

HMI.St9.EVInfo[40].dTime := PRG_Diagnostic.fbEVSt09[4].Q_tElapsedTimeFwd;		
HMI.St9.EVInfo[41].dTime := PRG_Diagnostic.fbEVSt09[4].Q_tElapsedTimeBwd;
END_ACTION

ACTION A_09_EVDiagnostic:
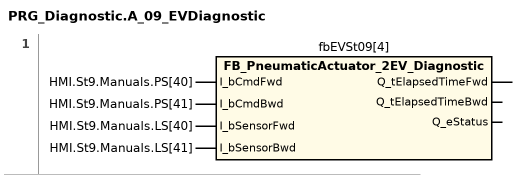
// NETWORK 1
fbEVSt09[4](
    I_bCmdFwd := HMI.St9.Manuals.PS[40],
    I_bCmdBwd := HMI.St9.Manuals.PS[41],
    I_bSensorFwd := HMI.St9.Manuals.LS[40],
    I_bSensorBwd := HMI.St9.Manuals.LS[41]); // FB_PneumaticActuator_2EV_Diagnostic
END_ACTION

ACTION A_10_Alarms:
FOR i:= 0 TO CNC.NUM_MAX_STATION_ALARMS -1 DO 
	StAlr[10][i] := PRG_EventManagement._PMCEventCollectors._CheckFanucPMCActiveAlarmList_St10_Alr._PMCEvents[i].bRaised;
END_FOR

HMI.St10.EVInfo[40].Error := PRG_Diagnostic.fbEVSt10[4].Q_eStatus = eEV_Status.MovingForward   AND StAlr[10][0];		
HMI.St10.EVInfo[41].Error := PRG_Diagnostic.fbEVSt10[4].Q_eStatus = eEV_Status.MovingBackward  AND StAlr[10][0];
HMI.St10.EVInfo[40].Error := PRG_Diagnostic.fbEVSt10[11].Q_eStatus = eEV_Status.MovingForward  AND StAlr[10][0];
HMI.St10.EVInfo[41].Error := PRG_Diagnostic.fbEVSt10[11].Q_eStatus = eEV_Status.MovingBackward AND StAlr[10][0]; 
                                                  
HMI.St10.EVInfo[54].dTime := PRG_Diagnostic.fbEVSt10[4].Q_tElapsedTimeFwd;		
HMI.St10.EVInfo[55].dTime := PRG_Diagnostic.fbEVSt10[4].Q_tElapsedTimeBwd;
HMI.St10.EVInfo[54].dTime := PRG_Diagnostic.fbEVSt10[11].Q_tElapsedTimeFwd;
HMI.St10.EVInfo[55].dTime := PRG_Diagnostic.fbEVSt10[11].Q_tElapsedTimeBwd;
END_ACTION

ACTION A_10_EVDiagnostic:
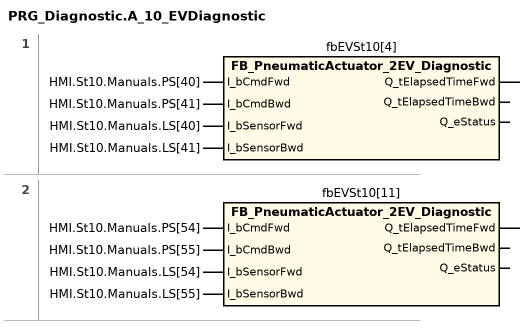
// NETWORK 1
fbEVSt10[4](
    I_bCmdFwd := HMI.St10.Manuals.PS[40],
    I_bCmdBwd := HMI.St10.Manuals.PS[41],
    I_bSensorFwd := HMI.St10.Manuals.LS[40],
    I_bSensorBwd := HMI.St10.Manuals.LS[41]); // FB_PneumaticActuator_2EV_Diagnostic

// NETWORK 2
fbEVSt10[11](
    I_bCmdFwd := HMI.St10.Manuals.PS[54],
    I_bCmdBwd := HMI.St10.Manuals.PS[55],
    I_bSensorFwd := HMI.St10.Manuals.LS[54],
    I_bSensorBwd := HMI.St10.Manuals.LS[55]); // FB_PneumaticActuator_2EV_Diagnostic
END_ACTION

ACTION A_11_Alarms:
FOR i:= 0 TO CNC.NUM_MAX_STATION_ALARMS -1 DO 
	StAlr[11][i] := PRG_EventManagement._PMCEventCollectors._CheckFanucPMCActiveAlarmList_St11_Alr._PMCEvents[i].bRaised;
END_FOR

HMI.St11.EVInfo[32].Error := PRG_Diagnostic.fbEVSt01[0].Q_eStatus = eEV_Status.MovingForward  AND StAlr[11][0];		
HMI.St11.EVInfo[33].Error := PRG_Diagnostic.fbEVSt01[0].Q_eStatus = eEV_Status.MovingBackward AND StAlr[11][0];
HMI.St11.EVInfo[34].Error := PRG_Diagnostic.fbEVSt01[1].Q_eStatus = eEV_Status.MovingForward  AND StAlr[11][0];
HMI.St11.EVInfo[35].Error := PRG_Diagnostic.fbEVSt01[1].Q_eStatus = eEV_Status.MovingBackward AND StAlr[11][0]; 

HMI.St11.EVInfo[32].dTime := PRG_Diagnostic.fbEVSt01[0].Q_tElapsedTimeFwd;		
HMI.St11.EVInfo[33].dTime := PRG_Diagnostic.fbEVSt01[0].Q_tElapsedTimeBwd;
HMI.St11.EVInfo[34].dTime := PRG_Diagnostic.fbEVSt01[1].Q_tElapsedTimeFwd;
HMI.St11.EVInfo[35].dTime := PRG_Diagnostic.fbEVSt01[1].Q_tElapsedTimeBwd;
END_ACTION

ACTION A_11_EVDiagnostic:
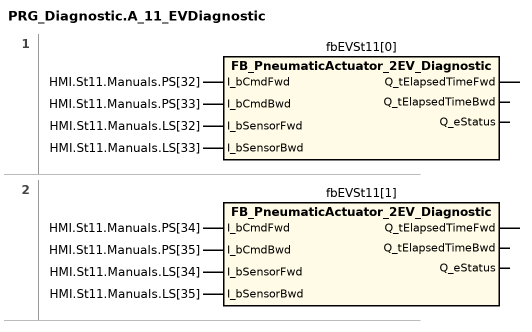
// NETWORK 1
fbEVSt11[0](
    I_bCmdFwd := HMI.St11.Manuals.PS[32],
    I_bCmdBwd := HMI.St11.Manuals.PS[33],
    I_bSensorFwd := HMI.St11.Manuals.LS[32],
    I_bSensorBwd := HMI.St11.Manuals.LS[33]); // FB_PneumaticActuator_2EV_Diagnostic

// NETWORK 2
fbEVSt11[1](
    I_bCmdFwd := HMI.St11.Manuals.PS[34],
    I_bCmdBwd := HMI.St11.Manuals.PS[35],
    I_bSensorFwd := HMI.St11.Manuals.LS[34],
    I_bSensorBwd := HMI.St11.Manuals.LS[35]); // FB_PneumaticActuator_2EV_Diagnostic
END_ACTION

ACTION A_12_Alarms:
FOR i:= 0 TO CNC.NUM_MAX_STATION_ALARMS -1 DO 
	StAlr[12][i] := PRG_EventManagement._PMCEventCollectors._CheckFanucPMCActiveAlarmList_St12_Alr._PMCEvents[i].bRaised;
END_FOR

HMI.St12.EVInfo[32].Error := PRG_Diagnostic.fbEVSt12[0].Q_eStatus = eEV_Status.MovingForward  AND StAlr[12][0];		
HMI.St12.EVInfo[33].Error := PRG_Diagnostic.fbEVSt12[0].Q_eStatus = eEV_Status.MovingBackward AND StAlr[12][0];
HMI.St12.EVInfo[34].Error := PRG_Diagnostic.fbEVSt12[1].Q_eStatus = eEV_Status.MovingForward  AND StAlr[12][0];
HMI.St12.EVInfo[35].Error := PRG_Diagnostic.fbEVSt12[1].Q_eStatus = eEV_Status.MovingBackward AND StAlr[12][0]; 
HMI.St12.EVInfo[36].Error := PRG_Diagnostic.fbEVSt12[2].Q_eStatus = eEV_Status.MovingForward  AND StAlr[12][0];		
HMI.St12.EVInfo[37].Error := PRG_Diagnostic.fbEVSt12[2].Q_eStatus = eEV_Status.MovingBackward AND StAlr[12][0];
HMI.St12.EVInfo[38].Error := PRG_Diagnostic.fbEVSt12[3].Q_eStatus = eEV_Status.MovingForward  AND StAlr[12][0];		
HMI.St12.EVInfo[39].Error := PRG_Diagnostic.fbEVSt12[3].Q_eStatus = eEV_Status.MovingBackward AND StAlr[12][0];
HMI.St12.EVInfo[40].Error := PRG_Diagnostic.fbEVSt12[4].Q_eStatus = eEV_Status.MovingForward  AND StAlr[12][0];		
HMI.St12.EVInfo[41].Error := PRG_Diagnostic.fbEVSt12[4].Q_eStatus = eEV_Status.MovingBackward AND StAlr[12][0]; 

HMI.St12.EVInfo[32].dTime := PRG_Diagnostic.fbEVSt12[0].Q_tElapsedTimeFwd;		
HMI.St12.EVInfo[33].dTime := PRG_Diagnostic.fbEVSt12[0].Q_tElapsedTimeBwd;
HMI.St12.EVInfo[34].dTime := PRG_Diagnostic.fbEVSt12[1].Q_tElapsedTimeFwd;
HMI.St12.EVInfo[35].dTime := PRG_Diagnostic.fbEVSt12[1].Q_tElapsedTimeBwd;
HMI.St12.EVInfo[36].dTime := PRG_Diagnostic.fbEVSt12[2].Q_tElapsedTimeFwd;		
HMI.St12.EVInfo[37].dTime := PRG_Diagnostic.fbEVSt12[2].Q_tElapsedTimeBwd;
HMI.St12.EVInfo[38].dTime := PRG_Diagnostic.fbEVSt12[3].Q_tElapsedTimeFwd;		
HMI.St12.EVInfo[39].dTime := PRG_Diagnostic.fbEVSt12[3].Q_tElapsedTimeBwd;
HMI.St12.EVInfo[40].dTime := PRG_Diagnostic.fbEVSt12[4].Q_tElapsedTimeFwd;		
HMI.St12.EVInfo[41].dTime := PRG_Diagnostic.fbEVSt12[4].Q_tElapsedTimeBwd;
END_ACTION

ACTION A_12_EVDiagnostic:
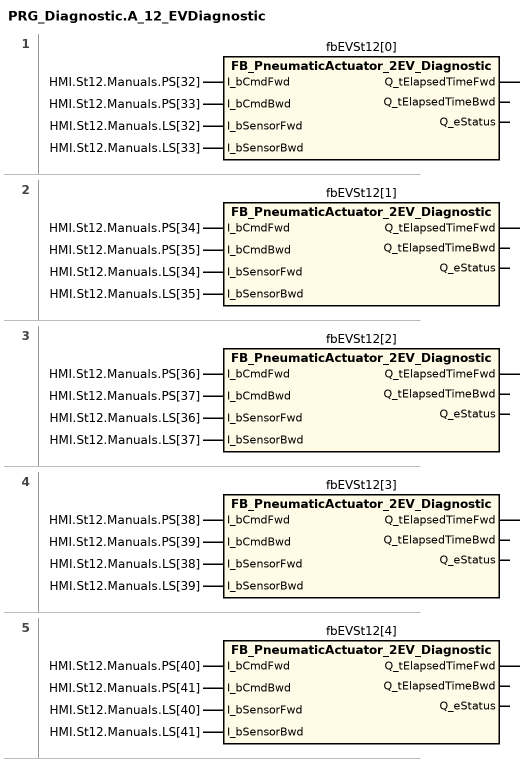
// NETWORK 1
fbEVSt12[0](
    I_bCmdFwd := HMI.St12.Manuals.PS[32],
    I_bCmdBwd := HMI.St12.Manuals.PS[33],
    I_bSensorFwd := HMI.St12.Manuals.LS[32],
    I_bSensorBwd := HMI.St12.Manuals.LS[33]); // FB_PneumaticActuator_2EV_Diagnostic

// NETWORK 2
fbEVSt12[1](
    I_bCmdFwd := HMI.St12.Manuals.PS[34],
    I_bCmdBwd := HMI.St12.Manuals.PS[35],
    I_bSensorFwd := HMI.St12.Manuals.LS[34],
    I_bSensorBwd := HMI.St12.Manuals.LS[35]); // FB_PneumaticActuator_2EV_Diagnostic

// NETWORK 3
fbEVSt12[2](
    I_bCmdFwd := HMI.St12.Manuals.PS[36],
    I_bCmdBwd := HMI.St12.Manuals.PS[37],
    I_bSensorFwd := HMI.St12.Manuals.LS[36],
    I_bSensorBwd := HMI.St12.Manuals.LS[37]); // FB_PneumaticActuator_2EV_Diagnostic

// NETWORK 4
fbEVSt12[3](
    I_bCmdFwd := HMI.St12.Manuals.PS[38],
    I_bCmdBwd := HMI.St12.Manuals.PS[39],
    I_bSensorFwd := HMI.St12.Manuals.LS[38],
    I_bSensorBwd := HMI.St12.Manuals.LS[39]); // FB_PneumaticActuator_2EV_Diagnostic

// NETWORK 5
fbEVSt12[4](
    I_bCmdFwd := HMI.St12.Manuals.PS[40],
    I_bCmdBwd := HMI.St12.Manuals.PS[41],
    I_bSensorFwd := HMI.St12.Manuals.LS[40],
    I_bSensorBwd := HMI.St12.Manuals.LS[41]); // FB_PneumaticActuator_2EV_Diagnostic
END_ACTION

ACTION A_13_Alarms:
FOR i:= 0 TO CNC.NUM_MAX_STATION_ALARMS -1 DO 
	StAlr[13][i] := PRG_EventManagement._PMCEventCollectors._CheckFanucPMCActiveAlarmList_St13_Alr._PMCEvents[i].bRaised;
END_FOR

HMI.St13.EVInfo[32].Error := PRG_Diagnostic.fbEVSt13[0].Q_eStatus = eEV_Status.MovingForward  AND StAlr[13][0];		
HMI.St13.EVInfo[33].Error := PRG_Diagnostic.fbEVSt13[0].Q_eStatus = eEV_Status.MovingBackward AND StAlr[13][0];
HMI.St13.EVInfo[34].Error := PRG_Diagnostic.fbEVSt13[1].Q_eStatus = eEV_Status.MovingForward  AND StAlr[13][0];
HMI.St13.EVInfo[35].Error := PRG_Diagnostic.fbEVSt13[1].Q_eStatus = eEV_Status.MovingBackward AND StAlr[13][0]; 
HMI.St13.EVInfo[36].Error := PRG_Diagnostic.fbEVSt13[2].Q_eStatus = eEV_Status.MovingForward  AND StAlr[13][0];		
HMI.St13.EVInfo[37].Error := PRG_Diagnostic.fbEVSt13[2].Q_eStatus = eEV_Status.MovingBackward AND StAlr[13][0]; 
HMI.St13.EVInfo[38].Error := PRG_Diagnostic.fbEVSt13[3].Q_eStatus = eEV_Status.MovingForward  AND StAlr[13][0];		
HMI.St13.EVInfo[39].Error := PRG_Diagnostic.fbEVSt13[3].Q_eStatus = eEV_Status.MovingBackward AND StAlr[13][0]; 

HMI.St13.EVInfo[32].dTime := PRG_Diagnostic.fbEVSt13[0].Q_tElapsedTimeFwd;		
HMI.St13.EVInfo[33].dTime := PRG_Diagnostic.fbEVSt13[0].Q_tElapsedTimeBwd;
HMI.St13.EVInfo[34].dTime := PRG_Diagnostic.fbEVSt13[1].Q_tElapsedTimeFwd;
HMI.St13.EVInfo[35].dTime := PRG_Diagnostic.fbEVSt13[1].Q_tElapsedTimeBwd;
HMI.St13.EVInfo[36].dTime := PRG_Diagnostic.fbEVSt13[2].Q_tElapsedTimeFwd;		
HMI.St13.EVInfo[37].dTime := PRG_Diagnostic.fbEVSt13[2].Q_tElapsedTimeBwd;
HMI.St13.EVInfo[38].dTime := PRG_Diagnostic.fbEVSt13[3].Q_tElapsedTimeFwd;		
HMI.St13.EVInfo[39].dTime := PRG_Diagnostic.fbEVSt13[3].Q_tElapsedTimeBwd;
END_ACTION

ACTION A_13_EVDiagnostic:
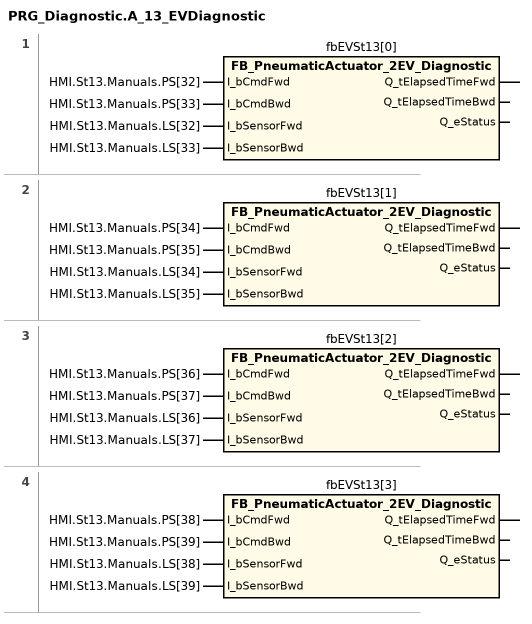
// NETWORK 1
fbEVSt13[0](
    I_bCmdFwd := HMI.St13.Manuals.PS[32],
    I_bCmdBwd := HMI.St13.Manuals.PS[33],
    I_bSensorFwd := HMI.St13.Manuals.LS[32],
    I_bSensorBwd := HMI.St13.Manuals.LS[33]); // FB_PneumaticActuator_2EV_Diagnostic

// NETWORK 2
fbEVSt13[1](
    I_bCmdFwd := HMI.St13.Manuals.PS[34],
    I_bCmdBwd := HMI.St13.Manuals.PS[35],
    I_bSensorFwd := HMI.St13.Manuals.LS[34],
    I_bSensorBwd := HMI.St13.Manuals.LS[35]); // FB_PneumaticActuator_2EV_Diagnostic

// NETWORK 3
fbEVSt13[2](
    I_bCmdFwd := HMI.St13.Manuals.PS[36],
    I_bCmdBwd := HMI.St13.Manuals.PS[37],
    I_bSensorFwd := HMI.St13.Manuals.LS[36],
    I_bSensorBwd := HMI.St13.Manuals.LS[37]); // FB_PneumaticActuator_2EV_Diagnostic

// NETWORK 4
fbEVSt13[3](
    I_bCmdFwd := HMI.St13.Manuals.PS[38],
    I_bCmdBwd := HMI.St13.Manuals.PS[39],
    I_bSensorFwd := HMI.St13.Manuals.LS[38],
    I_bSensorBwd := HMI.St13.Manuals.LS[39]); // FB_PneumaticActuator_2EV_Diagnostic
END_ACTION

END_PROGRAM

// ---- FBs/FB_PneumaticActuator_2EV_Diagnostic.TcPOU
FUNCTION_BLOCK FB_PneumaticActuator_2EV_Diagnostic
VAR_INPUT
	I_bCmdFwd					: BOOL;		// Comando avanti
	I_bCmdBwd					: BOOL;		// Comando indietro
	I_bSensorFwd				: BOOL;		// Sensore avanti
	I_bSensorBwd				: BOOL;		// Sensore indietro
END_VAR

VAR_OUTPUT
	Q_tElapsedTimeFwd			: UINT := 0;			// Durata movimento avanti
	Q_tElapsedTimeBwd			: UINT := 0;			// Durata movimento indietro
	//Q_tLastFwd					: UINT := 0;			// Durata ultimo movimento avanti
	//Q_tLastBwd					: UINT := 0;			// Durata ultimo movimento indietro
	Q_eStatus					: eEV_Status := eEV_Status.NotUsed; // Descrizione stato funzione
END_VAR

VAR
	_TON_TimerFwd				: TON;
	_TON_TimerBwd				: TON;
END_VAR

_TON_TimerFwd(IN := I_bCmdFwd AND NOT I_bSensorFwd, PT := T#99S);					
_TON_TimerBwd(IN := I_bCmdBwd AND NOT I_bSensorBwd, PT := T#99S);	

// Elapsed Time	
IF _TON_TimerBwd.IN THEN
	Q_tElapsedTimeBwd := TIME_TO_UINT(_TON_TimerBwd.ET);
END_IF
IF _TON_TimerFwd.IN THEN
	Q_tElapsedTimeFwd := TIME_TO_UINT(_TON_TimerFwd.ET);
END_IF
//IF I_bSensorFwd THEN
//	Q_tLastFwd := Q_tElapsedTimeFwd;
//ELSIF I_bSensorBwd THEN
//	Q_tLastBwd := Q_tElapsedTimeBwd;
//END_IF	
	
// Status
IF I_bCmdFwd AND NOT I_bSensorFwd THEN
	Q_eStatus := eEV_Status.MovingForward;
END_IF
IF I_bCmdBwd AND NOT I_bSensorBwd THEN
	Q_eStatus := eEV_Status.MovingBackward;
END_IF											
IF (Q_eStatus = eEV_Status.MovingBackward AND I_bSensorBwd) OR (Q_eStatus = eEV_Status.MovingForward AND I_bSensorFwd) THEN
	Q_eStatus := eEV_Status.MoveCompleted;
END_IF

END_FUNCTION_BLOCK

// ---- POUs/PRG_EventManagement.TcPOU
PROGRAM PRG_EventManagement
VAR
	// CNC  Alarms
	_FanucCNCActiveEventList AT %MB100: ARRAY [1..NUM_MAX_CNC_ACTIVE_EVENTS] OF U_FanucCNCEventEntry;
	_FanucCNCEventSourceList AT %MB21000 : ST_FanucCNCEventSourceList;
	_CheckFanucCNCActiveAlarmList : FB_CheckFanucCNCActiveEvents (CheckInterval := T#1S, 
																  CurrentCNCActiveEventList := _FanucCNCActiveEventList,
																  CNCEventSourceList := _FanucCNCEventSourceList);
																  
   _bEvents_InitDone 	: BOOL := FALSE;
   	iEvents_InitIndex 	: INT  := 0;
	iEvents_ClearIndex 	: INT  := 0;
	RTRIG_ClearEvents 	: R_TRIG;
	
	FanucPMCActiveAlarms AT %MB600: ARRAY [0..NUM_PMC_EVENTS / 8 - 1] OF BYTE;
	_PMCEventCollectors : FB_PMCEventCollectors(CheckInterval := T#1S, CurrentPMCActiveAlarmList := FanucPMCActiveAlarms);
	
	TestInt1 : UINT;
	TestInt2 : UINT;
	TestInt3 : UINT;
	
END_VAR


IF NOT _bEvents_InitDone THEN
	_PMCEventCollectors.Enabled := TRUE;
	_bEvents_InitDone := TRUE;
ELSE
	
// Monitor CNC Alarms
	_CheckFanucCNCActiveAlarmList(Enabled := TRUE);
	_PMCEventCollectors();
END_IF

END_PROGRAM

// ---- FBs/Events/FB_CheckFanucCNCActiveEvents.TcPOU
FUNCTION_BLOCK FB_CheckFanucCNCActiveEvents
VAR_INPUT
	Enabled : BOOL;
END_VAR
VAR

	{attribute 'hide'}
	_CNCEvents : ARRAY[0..NUM_CNC_EVENTS] OF FB_TcAlarm;

	{attribute 'hide'}
	_CurrentCNCActiveEventList : REFERENCE TO ARRAY [1..NUM_MAX_CNC_ACTIVE_EVENTS] OF U_FanucCNCEventEntry;

	{attribute 'hide'}
	_PreviousCNCActiveEventList : ARRAY [1..NUM_MAX_CNC_ACTIVE_EVENTS] OF U_FanucCNCEventEntry;
	
	{attribute 'hide'}
	_TcEventLogger : FB_TcEventLogger;	

	{attribute 'hide'}
	_CheckInterval : TIME;
	{attribute 'hide'}
	_CheckTimer : TON;
	
	{attribute 'hide'}
	_LastCreatedEventIndex : UINT := 0;	
	
	_CNCEventSourceList : REFERENCE TO ST_FanucCNCEventSourceList;

	_SourceInfoList : ARRAY [1..NUM_MAX_CNC_EVENT_SOURCES] OF FB_TcSourceInfo;
	
END_VAR

_CheckTimer();

IF Enabled AND (_CheckInterval > T#0MS) THEN
	IF _CheckTimer.Q THEN
		THIS^.UpdateActiveEventList();
		_CheckTimer.IN := FALSE;
	ELSE
		_CheckTimer.IN := TRUE;
	END_IF
ELSE
	_CheckTimer.IN := FALSE;
END_IF

METHOD PRIVATE BinarySearch : DINT;
VAR_INPUT
	_pTcEventEntry : POINTER TO TcEventEntry;
	_EventId : UDINT;
	_FirstIndex : UDINT;
	_LastIndex : UDINT;
END_VAR
VAR 
	_MiddleIndex : UDINT;
END_VAR
IF _FirstIndex = _LastIndex THEN
	IF _pTcEventEntry[_FirstIndex].nEventId = _EventId THEN
		BinarySearch := UDINT_TO_DINT(_FirstIndex);
	ELSE
		BinarySearch := -1;
	END_IF
ELSE
	_MiddleIndex := _FirstIndex + LREAL_TO_UDINT(FLOOR((_LastIndex - _FirstIndex) / 2));
	IF _pTcEventEntry[_MiddleIndex].nEventId >= _EventId THEN
		// Search on first half (recursive)
		BinarySearch := THIS^.BinarySearch(_pTcEventEntry, _EventId, _FirstIndex, _MiddleIndex);
	ELSE
		// Search on second half (recursive)
		BinarySearch := THIS^.BinarySearch(_pTcEventEntry, _EventId, _MiddleIndex + 1, _LastIndex);	
	END_IF
END_IF
END_METHOD

PROPERTY PUBLIC CheckInterval : TIME
GET
CheckInterval := _CheckInterval;
END_GET
SET
_CheckInterval := CheckInterval;
_CheckTimer.PT := _CheckInterval;
END_SET
END_PROPERTY

METHOD PUBLIC ClearAll : BOOL
VAR
	_TcEventFilter : FB_TcEventFilter;
	_i : BYTE;
	_EventClassInfo : ST_EventClassInfo;
	_NullGUID : GUID;
END_VAR
FOR _i := 0 TO 31 DO
	_EventClassInfo := GetEventClassInfo(_i);
	IF NOT GuidsEqualByVal(_EventClassInfo.GUID, _NullGUID) THEN
		_TcEventFilter.Clear().EventClass.EqualTo(_EventClassInfo.GUID);
		_TcEventLogger.ClearAlarms(0, FALSE, _TcEventFilter);
	END_IF
END_FOR
END_METHOD

METHOD FB_init : BOOL
VAR_INPUT
	bInitRetains : BOOL; // if TRUE, the retain variables are initialized (warm start / cold start)
	bInCopyCode : BOOL;  // if TRUE, the instance afterwards gets moved into the copy code (online change)
	CheckInterval : TIME;
	CurrentCNCActiveEventList : REFERENCE TO ARRAY [1..NUM_MAX_CNC_ACTIVE_EVENTS] OF U_FanucCNCEventEntry;
	CNCEventSourceList : REFERENCE TO ST_FanucCNCEventSourceList;
END_VAR
_CheckInterval := CheckInterval;
_CheckTimer.PT := _CheckInterval;

IF __ISVALIDREF(CurrentCNCActiveEventList) THEN
	_CurrentCNCActiveEventList REF= CurrentCNCActiveEventList;
END_IF

IF __ISVALIDREF(CNCEventSourceList) THEN
	_CNCEventSourceList REF= CNCEventSourceList;
END_IF

//InitSources();
END_METHOD

METHOD PRIVATE GetEventClassInfo : ST_EventClassInfo
VAR_INPUT
	ClassId : BYTE;
END_VAR
VAR
	_NullGUID : GUID;
END_VAR
CASE ClassId OF
	0:
		GetEventClassInfo.GUID := TC_EVENT_CLASSES.CNC_Alarms_SW;
		GetEventClassInfo.BaseAddress := ADR(TC_Events.CNC_Alarms_SW);
		GetEventClassInfo.Count := SIZEOF(TC_Events.CNC_Alarms_SW) / SIZEOF(TcEventEntry);
	1:
		GetEventClassInfo.GUID := TC_EVENT_CLASSES.CNC_Alarms_PW;
		GetEventClassInfo.BaseAddress := ADR(TC_Events.CNC_Alarms_PW);
		GetEventClassInfo.Count := SIZEOF(TC_Events.CNC_Alarms_PW) / SIZEOF(TcEventEntry);
	2:
		GetEventClassInfo.GUID := TC_EVENT_CLASSES.CNC_Alarms_IO;
		GetEventClassInfo.BaseAddress := ADR(TC_Events.CNC_Alarms_IO);
		GetEventClassInfo.Count := SIZEOF(TC_Events.CNC_Alarms_IO) / SIZEOF(TcEventEntry);
	3:
		GetEventClassInfo.GUID := TC_EVENT_CLASSES.CNC_Alarms_PS;
		GetEventClassInfo.BaseAddress := ADR(TC_Events.CNC_Alarms_PS);
		GetEventClassInfo.Count := SIZEOF(TC_Events.CNC_Alarms_PS) / SIZEOF(TcEventEntry);
	4:
		GetEventClassInfo.GUID := TC_EVENT_CLASSES.CNC_Alarms_OT;
		GetEventClassInfo.BaseAddress := ADR(TC_Events.CNC_Alarms_OT);
		GetEventClassInfo.Count := SIZEOF(TC_Events.CNC_Alarms_OT) / SIZEOF(TcEventEntry);
	5:
		GetEventClassInfo.GUID := TC_EVENT_CLASSES.CNC_Alarms_OH;
		GetEventClassInfo.BaseAddress := ADR(TC_Events.CNC_Alarms_OH);
		GetEventClassInfo.Count := SIZEOF(TC_Events.CNC_Alarms_OH) / SIZEOF(TcEventEntry);
	6:
		GetEventClassInfo.GUID := TC_EVENT_CLASSES.CNC_Alarms_SV;
		GetEventClassInfo.BaseAddress := ADR(TC_Events.CNC_Alarms_SV);
		GetEventClassInfo.Count := SIZEOF(TC_Events.CNC_Alarms_SV) / SIZEOF(TcEventEntry);
	7:
		GetEventClassInfo.GUID := TC_EVENT_CLASSES.CNC_Alarms_SR;
		GetEventClassInfo.BaseAddress := ADR(TC_Events.CNC_Alarms_SR);
		GetEventClassInfo.Count := SIZEOF(TC_Events.CNC_Alarms_SR) / SIZEOF(TcEventEntry);
	8:
		GetEventClassInfo.GUID := TC_EVENT_CLASSES.CNC_Alarms_MC;
		GetEventClassInfo.BaseAddress := ADR(TC_Events.CNC_Alarms_MC);
		GetEventClassInfo.Count := SIZEOF(TC_Events.CNC_Alarms_MC) / SIZEOF(TcEventEntry);
	9:
		GetEventClassInfo.GUID := TC_EVENT_CLASSES.CNC_Alarms_SP;
		GetEventClassInfo.BaseAddress := ADR(TC_Events.CNC_Alarms_SP);
		GetEventClassInfo.Count := SIZEOF(TC_Events.CNC_Alarms_SP) / SIZEOF(TcEventEntry);
	10:
		GetEventClassInfo.GUID := TC_EVENT_CLASSES.CNC_Alarms_DS;
		GetEventClassInfo.BaseAddress := ADR(TC_Events.CNC_Alarms_DS);
		GetEventClassInfo.Count := SIZEOF(TC_Events.CNC_Alarms_DS) / SIZEOF(TcEventEntry);
	11:
		GetEventClassInfo.GUID := TC_EVENT_CLASSES.CNC_Alarms_IE;
		GetEventClassInfo.BaseAddress := ADR(TC_Events.CNC_Alarms_IE);
		GetEventClassInfo.Count := SIZEOF(TC_Events.CNC_Alarms_IE) / SIZEOF(TcEventEntry);
//	12:
//		GetEventClassInfo.GUID := TC_EVENT_CLASSES.CNC_Alarms_BG;
//		GetEventClassInfo.BaseAddress := ADR(TC_Events.CNC_Alarms_BG);
//		GetEventClassInfo.Count := SIZEOF(TC_Events.CNC_Alarms_BG) / SIZEOF(TcEventEntry);
//	13:
//		GetEventClassInfo.GUID := TC_EVENT_CLASSES.CNC_Alarms_SN;
//		GetEventClassInfo.BaseAddress := ADR(TC_Events.CNC_Alarms_SN);
//		GetEventClassInfo.Count := SIZEOF(TC_Events.CNC_Alarms_SN) / SIZEOF(TcEventEntry);
//	15:
//		GetEventClassInfo.GUID := TC_EVENT_CLASSES.CNC_Alarms_EX;
//		GetEventClassInfo.BaseAddress := ADR(TC_Events.CNC_Alarms_EX);
//		GetEventClassInfo.Count := SIZEOF(TC_Events.CNC_Alarms_EX) / SIZEOF(TcEventEntry);
//	19:
//		GetEventClassInfo.GUID := TC_EVENT_CLASSES.CNC_Alarms_BG;
//		GetEventClassInfo.BaseAddress := ADR(TC_Events.CNC_Alarms_BG);
//		GetEventClassInfo.v := SIZEOF(TC_Events.CNC_Alarms_BG / SIZEOF(TcEventEntry));
	ELSE 
		GetEventClassInfo.GUID := _NullGUID;
		GetEventClassInfo.BaseAddress := 0;
		GetEventClassInfo.Count := 0;		
END_CASE
END_METHOD

METHOD PRIVATE GetSourceInfo : I_TcSourceInfo
VAR_INPUT
	SourceInfoId : DWORD;
END_VAR
VAR
	_iTcSourceInfo : I_TcSourceInfo;
	_Error : BOOL := FALSE;
	_i: UINT;
END_VAR
// Search for source
FOR _i := 1 TO NUM_MAX_CNC_EVENT_SOURCES DO
	IF SourceInfoId = _CNCEventSourceList.FanucCNCSources[_i].SourceId.Id THEN
		GetSourceInfo := _SourceInfoList[_i];
		RETURN;
	END_IF
END_FOR
END_METHOD

METHOD PRIVATE GetSourceInfoIndex : UINT
VAR_INPUT
	{attribute 'displaymode':='hex'}
	SourceInfoId : DWORD;
END_VAR
VAR
	_i: UINT;
END_VAR
// Search for source
FOR _i := 1 TO NUM_MAX_CNC_EVENT_SOURCES DO
	IF SourceInfoId = _CNCEventSourceList.FanucCNCSources[_i].SourceId.Id THEN
		GetSourceInfoIndex := _i;
		RETURN;
	END_IF
END_FOR
END_METHOD

METHOD PRIVATE InitSources : BOOL
VAR
	_i : UINT;
	_j : UINT;
	_k : UINT;
	_pTcEventEntry : POINTER TO TcEventEntry;
	_EventCount : UINT := 0;
	_SourceName : STRING;
	_SourceNameSB : clsStringBuilder;
END_VAR
IF __ISVALIDREF(_CNCEventSourceList) THEN
	FOR _i := 1 TO NUM_MAX_CNC_EVENT_SOURCES DO
		_SourceInfoList[_i].Clear();
		_SourceInfoList[_i].nId := _i;
		_SourceNameSB.Reset().Append(_CNCEventSourceList.FanucCNCSources[_i].CNCName).Append('.').Append(_CNCEventSourceList.FanucCNCSources[_i].PathName);
		_SourceName := _SourceNameSB.ToString();
		_SourceInfoList[_i].sName := _SourceName;
		//_SourceInfoList[_i].sName := CONCAT(_FanucCNCSourceList.FanucCNCSources[_i].CNCName, CONCAT('.', _FanucCNCSourceList.FanucCNCSources[_i].PathName));
	END_FOR
END_IF


//// Only for simulation
//FOR _i := 1 TO 10 DO
//	_FanucCNCSourceList.FanucCNCSources[_i].SourceId.Details.MainType := 1;
//	_FanucCNCSourceList.FanucCNCSources[_i].SourceId.Details.SubType := 0;
//	_FanucCNCSourceList.FanucCNCSources[_i].SourceId.Details.CNCNo := 1;
//	_FanucCNCSourceList.FanucCNCSources[_i].SourceId.Details.PathNo := UINT_TO_BYTE(_i);
//	_FanucCNCSourceList.FanucCNCSources[_i].CNCName := 'CNC1';
//	_FanucCNCSourceList.FanucCNCSources[_i].PathName := CONCAT('Path', TO_STRING(_i));
//	_FanucCNCSourceList.FanucCNCSources[_i].AxisNames[1] := CONCAT('X', TO_STRING(_i));
//	_FanucCNCSourceList.FanucCNCSources[_i].AxisNames[2] := CONCAT('Y', TO_STRING(_i));
//	_FanucCNCSourceList.FanucCNCSources[_i].AxisNames[3] := CONCAT('Z', TO_STRING(_i));
//	_SourceInfoList[_i].Clear();
//	_SourceInfoList[_i].nId := _i;
//	_SourceInfoList[_i].sName := CONCAT(_FanucCNCSourceList.FanucCNCSources[_i].CNCName, CONCAT('.', _FanucCNCSourceList.FanucCNCSources[_i].PathName));
//END_FOR
END_METHOD

METHOD PRIVATE SetParameters : BOOL
VAR_INPUT
	TcAlarm : REFERENCE TO FB_TcAlarm;
	FanucCNCEventSource : REFERENCE TO ST_FanucCNCEventSourceInfo;
	AxisMask : ST_FanucCNCEventAxesMask;
END_VAR
VAR
	_AxisList : STRING;
	_AxisListSB : clsStringBuilder;
END_VAR
_AxisList := '';
_AxisListSB.Reset();
TcAlarm.ipArguments.Clear();

IF __ISVALIDREF(FanucCNCEventSource) THEN

	IF AxisMask.Axis_1 THEN
		_AxisListSB.Append(FanucCNCEventSource.AxisNames[1]).Append(', ');
	END_IF
	IF AxisMask.Axis_2 THEN
		_AxisListSB.Append(FanucCNCEventSource.AxisNames[2]).Append(', ');
	END_IF
	IF AxisMask.Axis_3 THEN
		_AxisListSB.Append(FanucCNCEventSource.AxisNames[3]).Append(', ');
	END_IF
	IF AxisMask.Axis_4 THEN
		_AxisListSB.Append(FanucCNCEventSource.AxisNames[4]).Append(', ');
	END_IF
	IF AxisMask.Axis_5 THEN
		_AxisListSB.Append(FanucCNCEventSource.AxisNames[5]).Append(', ');
	END_IF
	IF AxisMask.Axis_6 THEN
		_AxisListSB.Append(FanucCNCEventSource.AxisNames[6]).Append(', ');
	END_IF
	IF AxisMask.Axis_7 THEN
		_AxisListSB.Append(FanucCNCEventSource.AxisNames[7]).Append(', ');
	END_IF
	IF AxisMask.Axis_8 THEN
		_AxisListSB.Append(FanucCNCEventSource.AxisNames[8]).Append(', ');
	END_IF
	
END_IF

IF	_AxisListSB.Length > 0 THEN
	_AxisListSB.Left(_AxisListSB.Length -2);
	_AxisList := _AxisListSB.ToString();
	TcAlarm.ipArguments.AddString(_AxisList);
END_IF
END_METHOD

METHOD PRIVATE UpdateActiveEventList : BOOL
VAR
	_i : UINT;
	_j : UINT;
	_Found : BOOL;	
	_TcAlarm : FB_TcAlarm;
	_refTcAlarm : REFERENCE TO FB_TcAlarm REF= _TcAlarm;
	_iTcSourceInfo : I_TcSourceInfo;
	_hr : HRESULT;
	_CNCNo : USINT;
	_PathNo : USINT;
	_pTcEventEntry : POINTER TO TcEventEntry;
	_EventIndex : DINT;
	_EventCount : UDINT;
	_EventClassId : BYTE;
	_EventId : UINT;
	_EventClassInfo : ST_EventClassInfo;
	_SourceInfoIndex : UINT;
END_VAR
// Check if previous and current memory areas for the list are same size
IF SIZEOF(_PreviousCNCActiveEventList) <> SIZEOF(_CurrentCNCActiveEventList) THEN
	UpdateActiveEventList := FALSE;
	RETURN;
END_IF

// Compare previous and current memory areas for differences
IF MEMCMP(ADR(_PreviousCNCActiveEventList), ADR(_CurrentCNCActiveEventList), SIZEOF(_CurrentCNCActiveEventList)) <> 0 THEN
	
	// In case of axes changing path during machining, the source needs to be updated at every change of active alarm list
	InitSources();

	// Check for events in previous list that are no longer active and clear them
	FOR _i := 1 TO NUM_MAX_CNC_ACTIVE_EVENTS DO
		IF _PreviousCNCActiveEventList[_i].Id <> 0 THEN
			_Found := FALSE;
			FOR _j := 1 TO NUM_MAX_CNC_ACTIVE_EVENTS DO
				IF _PreviousCNCActiveEventList[_i].Id = _CurrentCNCActiveEventList[_j].Id THEN
					_Found := TRUE;
					EXIT;
				END_IF
			END_FOR
			// If event previously active is no currently active: remove from list
			IF NOT _Found THEN
				_iTcSourceInfo := GetSourceInfo(_PreviousCNCActiveEventList[_i].Details.SourceInfo.Id);
				_EventClassId := _PreviousCNCActiveEventList[_i].Details.EventInfo.Details.Category;
				_EventId := _PreviousCNCActiveEventList[_i].Details.EventInfo.Details.No;
				_EventClassInfo := GetEventClassInfo(_EventClassId);
				IF _EventClassInfo.Count > 0 THEN 		// Event class contains no events
					_hr := _TcEventLogger.GetAlarm(_EventClassInfo.GUID, _EventId, _iTcSourceInfo, _refTcAlarm);
					IF SUCCEEDED(_hr) AND __ISVALIDREF(_refTcAlarm) THEN
						IF _refTcAlarm.bRaised THEN
							_refTcAlarm.Clear(0, TRUE);		// TODO: ResetConfirmation ??!!
						END_IF
					END_IF
				END_IF
			END_IF
		END_IF
	END_FOR
	
	// Check for events in current list that are not already active and raise them
	FOR _i := 1 TO NUM_MAX_CNC_ACTIVE_EVENTS DO
		IF _CurrentCNCActiveEventList[_i].Id <> 0 THEN
			_Found := FALSE;
			FOR _j := 1 TO NUM_MAX_CNC_ACTIVE_EVENTS DO
				IF _CurrentCNCActiveEventList[_i].Id = _PreviousCNCActiveEventList[_j].Id THEN
					_Found := TRUE;
					EXIT;
				END_IF
			END_FOR
			// If event currently active was not previously active: add to list
			IF NOT _Found THEN
				_SourceInfoIndex := GetSourceInfoIndex(_CurrentCNCActiveEventList[_i].Details.SourceInfo.Id);
				//_iTcSourceInfo := GetSourceInfo(_CurrentCNCActiveEventList[_i].Details.SourceInfo.Id);
				_iTcSourceInfo := _SourceInfoList[_SourceInfoIndex];
				_CNCNo := _CurrentCNCActiveEventList[_i].Details.SourceInfo.Details.CNCNo;
				_PathNo := _CurrentCNCActiveEventList[_i].Details.SourceInfo.Details.PathNo;
				_EventClassId := _CurrentCNCActiveEventList[_i].Details.EventInfo.Details.Category;
				_EventId := _CurrentCNCActiveEventList[_i].Details.EventInfo.Details.No;
				_EventClassInfo := GetEventClassInfo(_EventClassId);
				
				IF _EventClassInfo.Count > 0 THEN 		// Event class contains no events

					_hr := _TcEventLogger.GetAlarm(_EventClassInfo.GUID, _EventId, _iTcSourceInfo, _refTcAlarm);
					
					// Create event if not already created
					IF NOT SUCCEEDED(_hr) THEN
						_pTcEventEntry := _EventClassInfo.BaseAddress;
						_EventCount := _EventClassInfo.Count;
						_EventIndex := BinarySearch(_pTcEventEntry, _EventId, 0, _EventCount - 1);
						IF _EventIndex >= 0 THEN
							//CNC[_CNCNo].Paths[_PathNo].Alarms[_EventIndex].CreateEx(_pTcEventEntry[_EventIndex], FALSE, _iTcSourceInfo);	// TODO: NON SERVE!?! Eliminare?!
							_LastCreatedEventIndex := _LastCreatedEventIndex + 1;						
							_CNCEvents[_LastCreatedEventIndex].CreateEx(_pTcEventEntry[_EventIndex], FALSE, _iTcSourceInfo);
							_hr := _TcEventLogger.GetAlarm(_EventClassInfo.GUID, _EventId, _iTcSourceInfo, _refTcAlarm);
						END_IF
					END_IF
					
					IF SUCCEEDED(_hr) AND __ISVALIDREF(_refTcAlarm) THEN
						IF NOT _refTcAlarm.bRaised THEN
							_SourceInfoIndex := GetSourceInfoIndex(_CurrentCNCActiveEventList[_i].Details.SourceInfo.Id);
							SetParameters(_refTcAlarm, _CNCEventSourceList.FanucCNCSources[_SourceInfoIndex], _CurrentCNCActiveEventList[_i].Details.EventInfo.Details.AxesMask);
							_refTcAlarm.Raise(0);
						END_IF
					END_IF
					
				END_IF
					
			END_IF
		END_IF
	END_FOR
	
	// Update previous list with current list
	MEMCPY(ADR(_PreviousCNCActiveEventList), ADR(_CurrentCNCActiveEventList), SIZEOF(_CurrentCNCActiveEventList));

END_IF

UpdateActiveEventList := TRUE;
END_METHOD

END_FUNCTION_BLOCK

// ---- FBs/StringBuilder/clsStringBuilder.TcPOU
FUNCTION_BLOCK PUBLIC clsStringBuilder IMPLEMENTS  I_StringBuilder, I_LimitedStringBuilder
VAR
	{attribute 'hide'}
	_workString : STRING;
END_VAR

METHOD PUBLIC Append : I_StringBuilder // Append text to t current build string.
VAR_INPUT
	Text : STRING; //Text to append to current build string
END_VAR
_workString:= CONCAT(_WorkString, Text);
Append := THIS^;
END_METHOD

METHOD PUBLIC InsertAtLocation : I_StringBuilder
VAR_INPUT
	Text : STRING;
	Position : INT;
END_VAR
_WorkString := Tc2_Standard.INSERT(_WorkSTring, Text, Position);
InsertAtLocation := THIS^;
END_METHOD

METHOD PUBLIC Left : I_StringBuilder
VAR_INPUT
	Count	: INT;
END_VAR
_workString:= Tc2_Standard.LEFT(_WorkString, Count);
Left := THIS^;
END_METHOD

PROPERTY Length : INT
GET
Length := LEN(_workString);
END_GET
END_PROPERTY

METHOD PUBLIC Reset : I_LimitedStringBuilder // Reset current build string to an empty string.
_WorkString := '';
Reset := THIS^;
END_METHOD

METHOD Right : I_StringBuilder
VAR_INPUT
	Count	: INT;
END_VAR
_workString:= Tc2_Standard.RIGHT(_WorkString, Count);
Right := THIS^;
END_METHOD

METHOD PUBLIC ToString : STRING //Returns current build string.
ToString := _WorkString;
END_METHOD

END_FUNCTION_BLOCK

// ---- FBs/Events/FB_PMCEventCollectors.TcPOU
FUNCTION_BLOCK FB_PMCEventCollectors IMPLEMENTS I_EventDetailer
VAR

	//{attribute 'hide'}
	_Enabled : BOOL;

	{attribute 'hide'}
	_CheckInterval : TIME;
	
	{attribute 'hide'}
	_CheckTimer : TON;
	
	//{attribute 'hide'}
	_CurrentPMCActiveAlarmList : REFERENCE TO ARRAY [0..NUM_PMC_EVENTS / 8 - 1] OF BYTE;

	//{attribute 'hide'}
	_CurrentPMCActiveAlarmListCopy : ARRAY [0..NUM_PMC_EVENTS / 8 - 1] OF BYTE;

	//{attribute 'hide'}
	_PreviousPMCActiveAlarmList : ARRAY [0..NUM_PMC_EVENTS / 8 - 1] OF BYTE;

	// ###### ALARMS #####

	// PMC General Alarms 
	_CheckFanucPMCActiveAlarmList_Gen_Alr : FB_CheckFanucPMCActiveEvents (
						CheckInterval := T#0S, 
						CurrentPMCActiveAlarmList := _CurrentPMCActiveAlarmListCopy,
						PreviousPMCActiveAlarmList := _PreviousPMCActiveAlarmList,
						StartByte := 0,
						ByteLength := 60,
						SourceId := 99,
						SourceName := 'PMC',
						EventClass := ADR(TC_Events.AlrGeneral),
						EventDetailer := THIS^
						);
	
	// PMC St.0 (Manipulator) Alarms 
	_CheckFanucPMCActiveAlarmList_St00_Alr : FB_CheckFanucPMCActiveEvents (
						CheckInterval := T#0S, 
						CurrentPMCActiveAlarmList := _CurrentPMCActiveAlarmListCopy,
						PreviousPMCActiveAlarmList := _PreviousPMCActiveAlarmList,
						StartByte := 60,
						ByteLength := 40,
						SourceId := 100,
						SourceName := 'PMC',
						EventClass := ADR(TC_Events.Alr00),
						EventDetailer := THIS^
						);
	
	// PMC St.1 Alarms 
	_CheckFanucPMCActiveAlarmList_St01_Alr : FB_CheckFanucPMCActiveEvents (
						CheckInterval := T#0S, 
						CurrentPMCActiveAlarmList := _CurrentPMCActiveAlarmListCopy,
						PreviousPMCActiveAlarmList := _PreviousPMCActiveAlarmList,
						StartByte := 100,
						ByteLength := 10,
						SourceId := 101,
						SourceName := 'PMC',
						EventClass := ADR(TC_Events.Alr01),
						EventDetailer := THIS^
						);
	
	// PMC St.2 Alarms 
	_CheckFanucPMCActiveAlarmList_St02_Alr : FB_CheckFanucPMCActiveEvents (
						CheckInterval := T#0S, 
						CurrentPMCActiveAlarmList := _CurrentPMCActiveAlarmListCopy,
						PreviousPMCActiveAlarmList := _PreviousPMCActiveAlarmList,
						StartByte := 110,
						ByteLength := 10,
						SourceId := 102,
						SourceName := 'PMC',
						EventClass := ADR(TC_Events.Alr02),
						EventDetailer := THIS^
						);

	// PMC St.3 Alarms 
	_CheckFanucPMCActiveAlarmList_St03_Alr : FB_CheckFanucPMCActiveEvents (
						CheckInterval := T#0S, 
						CurrentPMCActiveAlarmList := _CurrentPMCActiveAlarmListCopy,
						PreviousPMCActiveAlarmList := _PreviousPMCActiveAlarmList,
						StartByte := 120,
						ByteLength := 10,
						SourceId := 103,
						SourceName := 'PMC',
						EventClass := ADR(TC_Events.Alr03),
						EventDetailer := THIS^
						);

	// PMC St.4 Alarms 
	_CheckFanucPMCActiveAlarmList_St04_Alr : FB_CheckFanucPMCActiveEvents (
						CheckInterval := T#0S, 
						CurrentPMCActiveAlarmList := _CurrentPMCActiveAlarmListCopy,
						PreviousPMCActiveAlarmList := _PreviousPMCActiveAlarmList,
						StartByte := 130,
						ByteLength := 10,
						SourceId := 104,
						SourceName := 'PMC',
						EventClass := ADR(TC_Events.Alr04),
						EventDetailer := THIS^
						);

	// PMC St.5 Alarms 
	_CheckFanucPMCActiveAlarmList_St05_Alr : FB_CheckFanucPMCActiveEvents (
						CheckInterval := T#0S, 
						CurrentPMCActiveAlarmList := _CurrentPMCActiveAlarmListCopy,
						PreviousPMCActiveAlarmList := _PreviousPMCActiveAlarmList,
						StartByte := 140,
						ByteLength := 10,
						SourceId := 105,
						SourceName := 'PMC',
						EventClass := ADR(TC_Events.Alr05),
						EventDetailer := THIS^
						);

	// PMC St.6 Alarms 
	_CheckFanucPMCActiveAlarmList_St06_Alr : FB_CheckFanucPMCActiveEvents (
						CheckInterval := T#0S, 
						CurrentPMCActiveAlarmList := _CurrentPMCActiveAlarmListCopy,
						PreviousPMCActiveAlarmList := _PreviousPMCActiveAlarmList,
						StartByte := 150,
						ByteLength := 10,
						SourceId := 106,
						SourceName := 'PMC',
						EventClass := ADR(TC_Events.Alr06),
						EventDetailer := THIS^
						);

	// PMC St.7 Alarms 
	_CheckFanucPMCActiveAlarmList_St07_Alr : FB_CheckFanucPMCActiveEvents (
						CheckInterval := T#0S, 
						CurrentPMCActiveAlarmList := _CurrentPMCActiveAlarmListCopy,
						PreviousPMCActiveAlarmList := _PreviousPMCActiveAlarmList,
						StartByte := 160,
						ByteLength := 10,
						SourceId := 107,
						SourceName := 'PMC',
						EventClass := ADR(TC_Events.Alr07),
						EventDetailer := THIS^
						);

	// PMC St.8 Alarms 
	_CheckFanucPMCActiveAlarmList_St08_Alr : FB_CheckFanucPMCActiveEvents (
						CheckInterval := T#0S, 
						CurrentPMCActiveAlarmList := _CurrentPMCActiveAlarmListCopy,
						PreviousPMCActiveAlarmList := _PreviousPMCActiveAlarmList,
						StartByte := 170,
						ByteLength := 10,
						SourceId := 108,
						SourceName := 'PMC',
						EventClass := ADR(TC_Events.Alr08),
						EventDetailer := THIS^
						);

	// PMC St.9 Alarms 
	_CheckFanucPMCActiveAlarmList_St09_Alr : FB_CheckFanucPMCActiveEvents (
						CheckInterval := T#0S, 
						CurrentPMCActiveAlarmList := _CurrentPMCActiveAlarmListCopy,
						PreviousPMCActiveAlarmList := _PreviousPMCActiveAlarmList,
						StartByte := 180,
						ByteLength := 10,
						SourceId := 109,
						SourceName := 'PMC',
						EventClass := ADR(TC_Events.Alr09),
						EventDetailer := THIS^
						);

	// PMC St.10 Alarms 
	_CheckFanucPMCActiveAlarmList_St10_Alr : FB_CheckFanucPMCActiveEvents (
						CheckInterval := T#0S, 
						CurrentPMCActiveAlarmList := _CurrentPMCActiveAlarmListCopy,
						PreviousPMCActiveAlarmList := _PreviousPMCActiveAlarmList,
						StartByte := 190,
						ByteLength := 10,
						SourceId := 110,
						SourceName := 'PMC',
						EventClass := ADR(TC_Events.Alr10),
						EventDetailer := THIS^
						);

	// PMC St.11 Alarms 
	_CheckFanucPMCActiveAlarmList_St11_Alr : FB_CheckFanucPMCActiveEvents (
						CheckInterval := T#0S, 
						CurrentPMCActiveAlarmList := _CurrentPMCActiveAlarmListCopy,
						PreviousPMCActiveAlarmList := _PreviousPMCActiveAlarmList,
						StartByte := 200,
						ByteLength := 10,
						SourceId := 111,
						SourceName := 'PMC',
						EventClass := ADR(TC_Events.Alr11),
						EventDetailer := THIS^
						);

	// PMC St.12 Alarms 
	_CheckFanucPMCActiveAlarmList_St12_Alr : FB_CheckFanucPMCActiveEvents (
						CheckInterval := T#0S, 
						CurrentPMCActiveAlarmList := _CurrentPMCActiveAlarmListCopy,
						PreviousPMCActiveAlarmList := _PreviousPMCActiveAlarmList,
						StartByte := 210,
						ByteLength := 10,
						SourceId := 112,
						SourceName := 'PMC',
						EventClass := ADR(TC_Events.Alr12),
						EventDetailer := THIS^
						);

	// PMC St.13 Alarms 
	_CheckFanucPMCActiveAlarmList_St13_Alr : FB_CheckFanucPMCActiveEvents (
						CheckInterval := T#0S, 
						CurrentPMCActiveAlarmList := _CurrentPMCActiveAlarmListCopy,
						PreviousPMCActiveAlarmList := _PreviousPMCActiveAlarmList,
						StartByte := 220,
						ByteLength := 10,
						SourceId := 113,
						SourceName := 'PMC',
						EventClass := ADR(TC_Events.Alr13),
						EventDetailer := THIS^
						);

//	// PMC St.14 Alarms 
//	_CheckFanucPMCActiveAlarmList_St14_Alr : FB_CheckFanucPMCActiveEvents (
//						CheckInterval := T#0S, 
//						CurrentPMCActiveAlarmList := _CurrentPMCActiveAlarmListCopy,
//						PreviousPMCActiveAlarmList := _PreviousPMCActiveAlarmList,
//						StartByte := 230,
//						ByteLength := 10,
//						SourceId := 114,
//						SourceName := 'PMC',
//						EventClass := ADR(TC_Events.Alr14),
//						EventDetailer := THIS^
//						);

//	// PMC St.15 Alarms 
//	_CheckFanucPMCActiveAlarmList_St15_Alr : FB_CheckFanucPMCActiveEvents (
//						CheckInterval := T#0S, 
//						CurrentPMCActiveAlarmList := _CurrentPMCActiveAlarmListCopy,
//						PreviousPMCActiveAlarmList := _PreviousPMCActiveAlarmList,
//						StartByte := 240,
//						ByteLength := 10,
//						SourceId := 115,
//						SourceName := 'PMC',
//						EventClass := ADR(TC_Events.Alr15),
//						EventDetailer := THIS^
//						);

//	// PMC St.16 Alarms 
//	_CheckFanucPMCActiveAlarmList_St16_Alr : FB_CheckFanucPMCActiveEvents (
//						CheckInterval := T#0S, 
//						CurrentPMCActiveAlarmList := _CurrentPMCActiveAlarmListCopy,
//						PreviousPMCActiveAlarmList := _PreviousPMCActiveAlarmList,
//						StartByte := 250,
//						ByteLength := 10,
//						SourceId := 116,
//						SourceName := 'PMC',
//						EventClass := ADR(TC_Events.Alr16),
//						EventDetailer := THIS^
//						);

//	// PMC St.17 Alarms 
//	_CheckFanucPMCActiveAlarmList_St17_Alr : FB_CheckFanucPMCActiveEvents (
//						CheckInterval := T#0S, 
//						CurrentPMCActiveAlarmList := _CurrentPMCActiveAlarmListCopy,
//						PreviousPMCActiveAlarmList := _PreviousPMCActiveAlarmList,
//						StartByte := 260,
//						ByteLength := 10,
//						SourceId := 117,
//						SourceName := 'PMC',
//						EventClass := ADR(TC_Events.Alr17),
//						EventDetailer := THIS^
//						);

//	// PMC St.18 Alarms 
//	_CheckFanucPMCActiveAlarmList_St18_Alr : FB_CheckFanucPMCActiveEvents (
//						CheckInterval := T#0S, 
//						CurrentPMCActiveAlarmList := _CurrentPMCActiveAlarmListCopy,
//						PreviousPMCActiveAlarmList := _PreviousPMCActiveAlarmList,
//						StartByte := 270,
//						ByteLength := 10,
//						SourceId := 118,
//						SourceName := 'PMC',
//						EventClass := ADR(TC_Events.Alr18),
//						EventDetailer := THIS^
//						);

//	// PMC St.19 Alarms 
//	_CheckFanucPMCActiveAlarmList_St19_Alr : FB_CheckFanucPMCActiveEvents (
//						CheckInterval := T#0S, 
//						CurrentPMCActiveAlarmList := _CurrentPMCActiveAlarmListCopy,
//						PreviousPMCActiveAlarmList := _PreviousPMCActiveAlarmList,
//						StartByte := 280,
//						ByteLength := 10,
//						SourceId := 119,
//						SourceName := 'St.19 ALR',
//						EventClass := ADR(TC_Events.Alr19),
//						EventDetailer := THIS^
//						);

						
	// ###### WARNINGS #####

	// PMC General Warnings
	_CheckFanucPMCActiveAlarmList_Gen_Wrn : FB_CheckFanucPMCActiveEvents (
						CheckInterval := T#0S, 
						CurrentPMCActiveAlarmList := _CurrentPMCActiveAlarmListCopy,
						PreviousPMCActiveAlarmList := _PreviousPMCActiveAlarmList,
						StartByte := 400,
						ByteLength := 10,
						SourceId := 99,
						SourceName := 'PMC',
						EventClass := ADR(TC_Events.WrnGeneral),
						EventDetailer := THIS^
						);
	
